C05452=1114.565,178.971,-64.399,-179.216,9.112,149.562
C05453=1114.569,178.722,-64.376,-179.219,9.109,149.562
C05454=1114.574,178.473,-64.352,-179.221,9.106,149.562
C05455=1114.579,178.224,-64.328,-179.223,9.103,149.562
C05456=1114.583,177.976,-64.304,-179.225,9.100,149.562
C05457=1114.588,177.727,-64.281,-179.228,9.097,149.562
C05458=1114.592,177.478,-64.257,-179.229,9.095,149.562
C05459=1114.597,177.229,-64.234,-179.232,9.091,149.562
C05460=1114.601,176.980,-64.210,-179.234,9.088,149.562
C05461=1114.606,176.732,-64.186,-179.236,9.086,149.561
C05462=1114.611,176.483,-64.163,-179.238,9.083,149.561
C05463=1114.615,176.233,-64.139,-179.241,9.079,149.561
C05464=1114.619,175.985,-64.115,-179.242,9.077,149.561
C05465=1114.624,175.736,-64.092,-179.245,9.074,149.561
C05466=1114.628,175.487,-64.068,-179.247,9.071,149.561
C05467=1114.633,175.238,-64.044,-179.249,9.068,149.561
C05468=1114.638,174.989,-64.021,-179.251,9.065,149.561
C05469=1114.642,174.740,-63.997,-179.253,9.062,149.561
C05470=1114.647,174.492,-63.973,-179.255,9.059,149.560
C05471=1114.651,174.243,-63.950,-179.258,9.056,149.560
C05472=1114.656,173.994,-63.927,-179.260,9.053,149.560
C05473=1114.661,173.745,-63.903,-179.262,9.050,149.560
C05474=1114.665,173.496,-63.879,-179.264,9.047,149.560
C05475=1114.670,173.247,-63.856,-179.267,9.044,149.560
C05476=1114.675,172.998,-63.833,-179.269,9.041,149.560
C05477=1114.678,172.749,-63.810,-179.271,9.038,149.560
C05478=1114.683,172.500,-63.786,-179.273,9.035,149.560
C05479=1114.687,172.287,-63.765,-179.275,9.032,149.560
C05480=1114.691,172.073,-63.745,-179.277,9.030,149.560
C05481=1114.695,171.860,-63.726,-179.278,9.027,149.559
C05482=1114.699,171.646,-63.706,-179.280,9.025,149.559
C05483=1114.703,171.432,-63.685,-179.282,9.023,149.559
C05484=1114.707,171.219,-63.666,-179.284,9.019,149.559
C05485=1114.711,171.005,-63.646,-179.286,9.017,149.559
C05486=1114.715,170.792,-63.626,-179.288,9.015,149.559
C05487=1114.719,170.543,-63.603,-179.290,9.011,149.559
C05488=1114.724,170.294,-63.579,-179.292,9.009,149.559
C05489=1114.728,170.045,-63.555,-179.295,9.006,149.559
C05490=1114.733,169.796,-63.532,-179.297,9.002,149.559
C05491=1114.737,169.548,-63.509,-179.299,8.999,149.559
C05492=1114.742,169.299,-63.486,-179.301,8.997,149.558
C05493=1114.747,169.050,-63.463,-179.303,8.993,149.558
C05494=1114.752,168.801,-63.439,-179.306,8.990,149.558
C05495=1114.756,168.552,-63.416,-179.308,8.987,149.558
C05496=1114.760,168.303,-63.393,-179.310,8.984,149.558
C05497=1114.765,168.054,-63.370,-179.312,8.981,149.558
C05498=1114.770,167.805,-63.347,-179.315,8.978,149.558
C05499=1114.774,167.557,-63.324,-179.317,8.975,149.558
C05500=1114.779,167.307,-63.301,-179.319,8.972,149.558
C05501=1114.784,167.059,-63.278,-179.321,8.969,149.558
C05502=1114.789,166.810,-63.255,-179.323,8.966,149.557
C05503=1114.793,166.561,-63.232,-179.326,8.963,149.557
C05504=1114.797,166.312,-63.209,-179.328,8.960,149.557
C05505=1114.802,166.063,-63.185,-179.330,8.957,149.557
C05506=1114.806,165.814,-63.163,-179.332,8.954,149.557
C05507=1114.811,165.566,-63.140,-179.335,8.951,149.557
C05508=1114.816,165.317,-63.116,-179.337,8.947,149.557
C05509=1114.820,165.067,-63.094,-179.339,8.945,149.557
C05510=1114.825,164.818,-63.071,-179.341,8.941,149.556
C05511=1114.830,164.569,-63.047,-179.343,8.938,149.556
C05512=1114.834,164.321,-63.025,-179.346,8.935,149.556
C05513=1114.839,164.072,-63.002,-179.348,8.932,149.556
C05514=1114.843,163.823,-62.980,-179.350,8.929,149.556
C05515=1114.848,163.574,-62.956,-179.352,8.926,149.556
C05516=1114.852,163.325,-62.934,-179.355,8.923,149.556
C05517=1114.857,163.076,-62.910,-179.357,8.919,149.556
C05518=1114.862,162.827,-62.888,-179.359,8.916,149.556
C05519=1114.866,162.579,-62.865,-179.362,8.913,149.555
C05520=1114.871,162.329,-62.842,-179.363,8.910,149.555
C05521=1114.875,162.080,-62.820,-179.366,8.907,149.555
C05522=1114.880,161.832,-62.797,-179.368,8.904,149.555
C05523=1114.884,161.583,-62.774,-179.370,8.901,149.555
C05524=1114.889,161.333,-62.751,-179.372,8.897,149.555
C05525=1114.893,161.085,-62.729,-179.375,8.894,149.555
C05526=1114.899,160.836,-62.706,-179.377,8.890,149.554
C05527=1114.903,160.587,-62.684,-179.379,8.888,149.554
C05528=1114.908,160.338,-62.660,-179.381,8.885,149.554
C05529=1114.912,160.089,-62.637,-179.383,8.882,149.554
C05530=1114.917,159.840,-62.615,-179.386,8.878,149.554
C05531=1114.921,159.592,-62.592,-179.388,8.875,149.554
C05532=1114.926,159.342,-62.570,-179.390,8.871,149.554
C05533=1114.930,159.093,-62.547,-179.393,8.868,149.554
C05534=1114.935,158.845,-62.525,-179.395,8.865,149.553
C05535=1114.939,158.631,-62.505,-179.397,8.862,149.553
C05536=1114.943,158.417,-62.486,-179.398,8.860,149.553
C05537=1114.947,158.203,-62.467,-179.401,8.857,149.553
C05538=1114.951,157.989,-62.448,-179.402,8.854,149.553
C05539=1114.955,157.776,-62.428,-179.405,8.851,149.553
C05540=1114.959,157.562,-62.409,-179.406,8.848,149.553
C05541=1114.963,157.349,-62.389,-179.408,8.846,149.553
C05542=1114.967,157.134,-62.370,-179.410,8.842,149.552
C05543=1114.972,156.886,-62.348,-179.413,8.839,149.552
C05544=1114.976,156.637,-62.326,-179.415,8.836,149.552
C05545=1114.981,156.388,-62.302,-179.417,8.833,149.552
C05546=1114.985,156.139,-62.281,-179.419,8.829,149.552
C05547=1114.990,155.890,-62.259,-179.421,8.826,149.552
C05548=1114.994,155.641,-62.235,-179.424,8.823,149.551
C05549=1114.999,155.392,-62.214,-179.425,8.820,149.551
C05550=1115.004,155.143,-62.191,-179.427,8.816,149.551
C05551=1115.008,154.894,-62.168,-179.430,8.813,149.551
C05552=1115.013,154.645,-62.146,-179.432,8.810,149.551
C05553=1115.017,154.396,-62.124,-179.435,8.805,149.551
C05554=1115.023,154.148,-62.101,-179.437,8.802,149.550
C05555=1115.027,153.898,-62.079,-179.439,8.799,149.550
C05556=1115.032,153.650,-62.058,-179.441,8.795,149.550
C05557=1115.036,153.400,-62.036,-179.443,8.792,149.550
C05558=1115.041,153.151,-62.012,-179.446,8.789,149.550
C05559=1115.046,152.903,-61.991,-179.448,8.785,149.550
C05560=1115.050,152.653,-61.969,-179.450,8.782,149.549
C05561=1115.055,152.405,-61.947,-179.452,8.778,149.549
C05562=1115.060,152.156,-61.923,-179.455,8.775,149.549
C05563=1115.064,151.907,-61.902,-179.457,8.772,149.549
C05564=1115.069,151.658,-61.880,-179.459,8.768,149.549
C05565=1115.074,151.409,-61.858,-179.461,8.765,149.548
C05566=1115.078,151.160,-61.836,-179.463,8.761,149.548
C05567=1115.083,150.910,-61.813,-179.466,8.758,149.548
C05568=1115.088,150.661,-61.792,-179.468,8.755,149.548
C05569=1115.092,150.412,-61.770,-179.470,8.750,149.548
C05570=1115.097,150.164,-61.747,-179.472,8.747,149.547
C05571=1115.101,149.915,-61.725,-179.475,8.743,149.547
C05572=1115.106,149.666,-61.704,-179.477,8.740,149.547
C05573=1115.111,149.417,-61.682,-179.479,8.736,149.547
C05574=1115.116,149.168,-61.659,-179.481,8.733,149.546
C05575=1115.120,148.919,-61.638,-179.483,8.729,149.546
C05576=1115.125,148.670,-61.615,-179.485,8.726,149.546
C05577=1115.130,148.421,-61.594,-179.488,8.722,149.546
C05578=1115.134,148.172,-61.572,-179.490,8.718,149.545
C05579=1115.139,147.923,-61.550,-179.492,8.715,149.545
C05580=1115.143,147.674,-61.528,-179.494,8.711,149.545
C05581=1115.148,147.425,-61.506,-179.496,8.708,149.545
C05582=1115.152,147.176,-61.484,-179.499,8.704,149.544
C05583=1115.157,146.927,-61.463,-179.501,8.700,149.544
C05584=1115.162,146.677,-61.441,-179.503,8.697,149.544
C05585=1115.166,146.429,-61.420,-179.505,8.693,149.544
C05586=1115.171,146.180,-61.398,-179.507,8.690,149.544
C05587=1115.176,145.931,-61.376,-179.510,8.685,149.543
C05588=1115.180,145.682,-61.354,-179.512,8.682,149.543
C05589=1115.185,145.433,-61.332,-179.514,8.678,149.543
C05590=1115.190,145.184,-61.310,-179.516,8.675,149.543
C05591=1115.194,144.970,-61.291,-179.518,8.671,149.542
C05592=1115.198,144.756,-61.274,-179.519,8.668,149.542
C05593=1115.202,144.542,-61.255,-179.520,8.666,149.542
C05594=1115.206,144.329,-61.237,-179.521,8.662,149.541
C05595=1115.210,144.114,-61.218,-179.523,8.660,149.541
C05596=1115.213,143.901,-61.199,-179.524,8.657,149.541
C05597=1115.218,143.687,-61.180,-179.525,8.654,149.540
C05598=1115.221,143.473,-61.162,-179.527,8.651,149.540
C05599=1115.226,143.225,-61.140,-179.529,8.648,149.540
C05600=1115.231,142.975,-61.119,-179.531,8.644,149.539
C05601=1115.236,142.726,-61.097,-179.532,8.641,149.539
C05602=1115.241,142.477,-61.076,-179.534,8.637,149.539
C05603=1115.245,142.227,-61.054,-179.536,8.634,149.539
C05604=1115.250,141.979,-61.033,-179.537,8.631,149.538
C05605=1115.255,141.730,-61.011,-179.539,8.627,149.538
C05606=1115.259,141.480,-60.990,-179.540,8.623,149.537
C05607=1115.264,141.232,-60.968,-179.542,8.621,149.537
C05608=1115.268,140.983,-60.947,-179.544,8.617,149.537
C05609=1115.273,140.733,-60.925,-179.545,8.614,149.537
C05610=1115.278,140.485,-60.904,-179.547,8.610,149.536
C05611=1115.283,140.236,-60.882,-179.549,8.607,149.536
C05612=1115.287,139.986,-60.861,-179.550,8.604,149.536
C05613=1115.291,139.738,-60.840,-179.552,8.600,149.535
C05614=1115.297,139.488,-60.819,-179.554,8.597,149.535
C05615=1115.301,139.240,-60.797,-179.555,8.594,149.535
C05616=1115.306,138.990,-60.775,-179.557,8.590,149.534
C05617=1115.310,138.741,-60.755,-179.559,8.587,149.534
C05618=1115.315,138.493,-60.733,-179.560,8.583,149.534
C05619=1115.320,138.243,-60.712,-179.562,8.580,149.533
C05620=1115.324,137.994,-60.690,-179.563,8.577,149.533
C05621=1115.329,137.745,-60.669,-179.565,8.573,149.533
C05622=1115.334,137.497,-60.648,-179.567,8.570,149.533
C05623=1115.338,137.247,-60.626,-179.568,8.567,149.532
C05624=1115.343,136.998,-60.605,-179.570,8.563,149.532
C05625=1115.348,136.749,-60.584,-179.572,8.560,149.532
C05626=1115.353,136.500,-60.563,-179.573,8.557,149.531
C05627=1115.357,136.250,-60.541,-179.575,8.553,149.531
C05628=1115.361,136.002,-60.520,-179.578,8.550,149.531
C05629=1115.366,135.753,-60.499,-179.579,8.547,149.530
C05630=1115.372,135.504,-60.478,-179.581,8.543,149.530
C05631=1115.376,135.255,-60.457,-179.583,8.540,149.530
C05632=1115.380,135.005,-60.436,-179.584,8.537,149.529
C05633=1115.385,134.757,-60.414,-179.586,8.533,149.529
C05634=1115.390,134.507,-60.393,-179.587,8.530,149.529
C05635=1115.395,134.258,-60.373,-179.589,8.527,149.529
C05636=1115.400,134.010,-60.351,-179.591,8.523,149.528
C05637=1115.404,133.760,-60.330,-179.592,8.520,149.528
C05638=1115.409,133.511,-60.310,-179.594,8.516,149.528
C05639=1115.414,133.262,-60.288,-179.596,8.513,149.527
C05640=1115.418,133.013,-60.267,-179.598,8.510,149.527
C05641=1115.423,132.764,-60.247,-179.599,8.506,149.527
C05642=1115.428,132.515,-60.225,-179.601,8.503,149.526
C05643=1115.432,132.266,-60.204,-179.603,8.500,149.526
C05644=1115.437,132.017,-60.183,-179.605,8.497,149.526
C05645=1115.441,131.768,-60.163,-179.606,8.493,149.526
C05646=1115.446,131.519,-60.141,-179.608,8.490,149.525
C05647=1115.451,131.305,-60.124,-179.609,8.487,149.525
C05648=1115.454,131.091,-60.106,-179.611,8.484,149.525
C05649=1115.459,130.877,-60.087,-179.613,8.481,149.525
C05650=1115.463,130.663,-60.069,-179.614,8.478,149.524
C05651=1115.467,130.449,-60.052,-179.616,8.476,149.524
C05652=1115.470,130.235,-60.034,-179.617,8.473,149.524
C05653=1115.474,130.021,-60.016,-179.618,8.470,149.524
C05654=1115.479,129.807,-59.998,-179.620,8.467,149.523
C05655=1115.484,129.558,-59.978,-179.622,8.464,149.523
C05656=1115.488,129.309,-59.956,-179.624,8.460,149.523
C05657=1115.493,129.060,-59.935,-179.625,8.457,149.522
C05658=1115.498,128.811,-59.914,-179.627,8.454,149.522
C05659=1115.502,128.562,-59.894,-179.629,8.450,149.522
C05660=1115.507,128.312,-59.873,-179.630,8.447,149.522
C05661=1115.512,128.063,-59.853,-179.632,8.444,149.521
C05662=1115.517,127.814,-59.832,-179.634,8.440,149.521
C05663=1115.521,127.565,-59.811,-179.635,8.437,149.521
C05664=1115.527,127.316,-59.790,-179.637,8.434,149.521
C05665=1115.531,127.067,-59.770,-179.639,8.430,149.520
C05666=1115.535,126.818,-59.750,-179.641,8.427,149.520
C05667=1115.541,126.569,-59.729,-179.643,8.424,149.520
C05668=1115.545,126.320,-59.708,-179.645,8.420,149.520
C05669=1115.550,126.071,-59.687,-179.646,8.418,149.519
C05670=1115.555,125.822,-59.667,-179.648,8.414,149.519
C05671=1115.559,125.573,-59.647,-179.650,8.410,149.519
C05672=1115.564,125.323,-59.626,-179.652,8.407,149.518
C05673=1115.569,125.075,-59.605,-179.653,8.404,149.518
C05674=1115.573,124.825,-59.584,-179.655,8.400,149.518
C05675=1115.578,124.576,-59.563,-179.657,8.397,149.518
C05676=1115.582,124.327,-59.543,-179.658,8.394,149.517
C05677=1115.587,124.077,-59.522,-179.660,8.390,149.517
C05678=1115.592,123.828,-59.502,-179.662,8.386,149.517
C05679=1115.596,123.580,-59.481,-179.664,8.384,149.516
C05680=1115.601,123.330,-59.460,-179.666,8.380,149.516
C05681=1115.606,123.081,-59.440,-179.668,8.377,149.516
C05682=1115.611,122.833,-59.420,-179.669,8.373,149.516
C05683=1115.616,122.583,-59.400,-179.671,8.370,149.515
C05684=1115.621,122.334,-59.379,-179.673,8.367,149.515
C05685=1115.625,122.085,-59.359,-179.675,8.363,149.515
C05686=1115.630,121.836,-59.339,-179.676,8.360,149.515
C05687=1115.635,121.587,-59.318,-179.678,8.357,149.514
C05688=1115.640,121.338,-59.298,-179.680,8.353,149.514
C05689=1115.644,121.089,-59.278,-179.682,8.350,149.514
C05690=1115.648,120.840,-59.257,-179.684,8.347,149.514
C05691=1115.654,120.590,-59.236,-179.685,8.343,149.513
C05692=1115.658,120.341,-59.216,-179.687,8.339,149.513
C05693=1115.663,120.092,-59.196,-179.689,8.337,149.513
C05694=1115.667,119.843,-59.176,-179.691,8.333,149.512
C05695=1115.672,119.594,-59.155,-179.692,8.329,149.512
C05696=1115.677,119.344,-59.135,-179.694,8.326,149.512
C05697=1115.682,119.095,-59.115,-179.696,8.323,149.512
C05698=1115.687,118.847,-59.095,-179.698,8.320,149.511
C05699=1115.691,118.597,-59.075,-179.700,8.316,149.511
C05700=1115.696,118.348,-59.055,-179.702,8.312,149.511
C05701=1115.701,118.099,-59.034,-179.703,8.310,149.510
C05702=1115.706,117.850,-59.014,-179.705,8.306,149.510
C05703=1115.710,117.636,-58.997,-179.707,8.303,149.510
C05704=1115.714,117.422,-58.979,-179.709,8.300,149.510
C05705=1115.717,117.208,-58.962,-179.710,8.297,149.509
C05706=1115.721,116.994,-58.945,-179.711,8.294,149.509
C05707=1115.726,116.780,-58.928,-179.712,8.291,149.509
C05708=1115.730,116.566,-58.911,-179.714,8.289,149.509
C05709=1115.734,116.351,-58.893,-179.716,8.285,149.508
C05710=1115.738,116.137,-58.876,-179.717,8.282,149.508
C05711=1115.743,115.888,-58.856,-179.719,8.279,149.508
C05712=1115.748,115.640,-58.836,-179.720,8.276,149.508
C05713=1115.753,115.390,-58.816,-179.722,8.272,149.507
C05714=1115.757,115.141,-58.796,-179.725,8.269,149.507
C05715=1115.762,114.892,-58.776,-179.727,8.265,149.507
C05716=1115.766,114.643,-58.756,-179.728,8.261,149.506
C05717=1115.771,114.393,-58.736,-179.730,8.259,149.506
C05718=1115.776,114.145,-58.716,-179.732,8.255,149.506
C05719=1115.781,113.895,-58.697,-179.734,8.252,149.506
C05720=1115.786,113.646,-58.676,-179.735,8.248,149.505
C05721=1115.791,113.396,-58.656,-179.737,8.244,149.505
C05722=1115.795,113.147,-58.636,-179.739,8.242,149.505
C05723=1115.800,112.899,-58.616,-179.740,8.238,149.504
C05724=1115.805,112.649,-58.597,-179.743,8.234,149.504
C05725=1115.810,112.400,-58.576,-179.745,8.231,149.504
C05726=1115.814,112.151,-58.557,-179.746,8.227,149.504
C05727=1115.820,111.902,-58.537,-179.748,8.224,149.503
C05728=1115.824,111.653,-58.517,-179.750,8.221,149.503
C05729=1115.829,111.403,-58.497,-179.751,8.217,149.503
C05730=1115.833,111.154,-58.477,-179.753,8.213,149.502
C05731=1115.839,110.905,-58.458,-179.755,8.210,149.502
C05732=1115.843,110.656,-58.439,-179.758,8.206,149.502
C05733=1115.847,110.406,-58.419,-179.760,8.203,149.502
C05734=1115.852,110.158,-58.399,-179.762,8.198,149.502
C05735=1115.857,109.909,-58.379,-179.764,8.195,149.501
C05736=1115.862,109.659,-58.360,-179.766,8.191,149.501
C05737=1115.867,109.410,-58.340,-179.768,8.188,149.501
C05738=1115.872,109.161,-58.320,-179.770,8.184,149.500
C05739=1115.876,108.912,-58.300,-179.773,8.180,149.500
C05740=1115.881,108.662,-58.281,-179.775,8.176,149.500
C05741=1115.887,108.413,-58.261,-179.776,8.172,149.500
C05742=1115.890,108.165,-58.242,-179.778,8.169,149.499
C05743=1115.895,107.915,-58.222,-179.781,8.165,149.499
C05744=1115.900,107.666,-58.203,-179.783,8.161,149.499
C05745=1115.905,107.417,-58.183,-179.785,8.157,149.498
C05746=1115.910,107.167,-58.163,-179.787,8.154,149.498
C05747=1115.915,106.918,-58.144,-179.788,8.150,149.498
C05748=1115.919,106.669,-58.125,-179.791,8.146,149.498
C05749=1115.924,106.419,-58.105,-179.793,8.142,149.497
C05750=1115.929,106.171,-58.085,-179.795,8.138,149.497
C05751=1115.934,105.922,-58.066,-179.797,8.135,149.497
C05752=1115.938,105.672,-58.047,-179.799,8.131,149.496
C05753=1115.943,105.423,-58.027,-179.801,8.127,149.496
C05754=1115.948,105.174,-58.008,-179.803,8.124,149.496
C05755=1115.953,104.925,-57.988,-179.804,8.120,149.495
C05756=1115.957,104.676,-57.969,-179.807,8.116,149.495
C05757=1115.962,104.426,-57.950,-179.808,8.112,149.495
C05758=1115.967,104.177,-57.930,-179.811,8.108,149.494
C05759=1115.971,103.963,-57.914,-179.812,8.105,149.494
C05760=1115.976,103.749,-57.897,-179.814,8.102,149.494
C05761=1115.980,103.534,-57.881,-179.815,8.099,149.494
C05762=1115.984,103.321,-57.864,-179.817,8.095,149.493
C05763=1115.988,103.107,-57.847,-179.818,8.092,149.493
C05764=1115.992,102.892,-57.831,-179.820,8.089,149.493
C05765=1115.996,102.678,-57.815,-179.822,8.085,149.492
C05766=1116.000,102.464,-57.798,-179.823,8.082,149.492
C05767=1116.005,102.214,-57.779,-179.825,8.078,149.492
C05768=1116.010,101.966,-57.760,-179.827,8.075,149.491
C05769=1116.015,101.716,-57.740,-179.828,8.071,149.491
C05770=1116.020,101.467,-57.721,-179.830,8.067,149.491
C05771=1116.024,101.218,-57.702,-179.832,8.064,149.490
C05772=1116.029,100.969,-57.683,-179.834,8.059,149.490
C05773=1116.034,100.719,-57.664,-179.836,8.055,149.489
C05774=1116.039,100.470,-57.645,-179.837,8.051,149.489
C05775=1116.044,100.221,-57.625,-179.840,8.048,149.489
C05776=1116.048,99.972,-57.607,-179.841,8.044,149.488
C05777=1116.053,99.723,-57.587,-179.843,8.040,149.488
C05778=1116.058,99.474,-57.569,-179.844,8.036,149.488
C05779=1116.063,99.224,-57.549,-179.846,8.032,149.487
C05780=1116.067,98.975,-57.531,-179.848,8.029,149.487
C05781=1116.072,98.725,-57.512,-179.850,8.025,149.486
C05782=1116.078,98.476,-57.493,-179.851,8.021,149.486
C05783=1116.082,98.227,-57.473,-179.853,8.017,149.486
C05784=1116.087,97.978,-57.454,-179.854,8.013,149.485
C05785=1116.091,97.728,-57.436,-179.856,8.009,149.485
C05786=1116.097,97.480,-57.417,-179.858,8.006,149.484
C05787=1116.101,97.230,-57.397,-179.860,8.002,149.484
C05788=1116.106,96.981,-57.379,-179.861,7.998,149.484
C05789=1116.110,96.732,-57.360,-179.863,7.994,149.483
C05790=1116.116,96.482,-57.341,-179.864,7.990,149.483
C05791=1116.121,96.234,-57.323,-179.866,7.986,149.482
C05792=1116.125,95.984,-57.304,-179.868,7.982,149.482
C05793=1116.130,95.735,-57.285,-179.869,7.978,149.481
C05794=1116.134,95.486,-57.266,-179.871,7.974,149.481
C05795=1116.140,95.236,-57.247,-179.872,7.971,149.481
C05796=1116.144,94.987,-57.229,-179.874,7.967,149.480
C05797=1116.150,94.737,-57.210,-179.875,7.964,149.480
C05798=1116.154,94.489,-57.191,-179.877,7.960,149.479
C05799=1116.159,94.239,-57.171,-179.878,7.956,149.479
C05800=1116.164,93.990,-57.153,-179.880,7.952,149.478
C05801=1116.168,93.741,-57.135,-179.881,7.948,149.478
C05802=1116.173,93.491,-57.116,-179.883,7.944,149.478
C05803=1116.178,93.242,-57.098,-179.885,7.940,149.477
C05804=1116.183,92.994,-57.079,-179.886,7.936,149.476
C05805=1116.188,92.743,-57.060,-179.887,7.932,149.476
C05806=1116.193,92.495,-57.041,-179.889,7.928,149.476
C05807=1116.198,92.245,-57.023,-179.890,7.925,149.475
C05808=1116.202,91.996,-57.004,-179.892,7.921,149.475
C05809=1116.207,91.747,-56.986,-179.893,7.917,149.474
C05810=1116.213,91.497,-56.967,-179.895,7.913,149.474
C05811=1116.217,91.248,-56.948,-179.896,7.909,149.473
C05812=1116.222,90.999,-56.930,-179.897,7.905,149.473
C05813=1116.226,90.750,-56.911,-179.899,7.901,149.472
C05814=1116.231,90.500,-56.893,-179.900,7.898,149.472
C05815=1116.235,90.286,-56.876,-179.902,7.894,149.472
C05816=1116.240,90.072,-56.861,-179.903,7.891,149.471
C05817=1116.244,89.858,-56.845,-179.904,7.888,149.471
C05818=1116.248,89.644,-56.829,-179.905,7.885,149.470
C05819=1116.252,89.429,-56.813,-179.906,7.881,149.470
C05820=1116.256,89.215,-56.797,-179.907,7.878,149.469
C05821=1116.261,89.001,-56.781,-179.908,7.875,149.469
C05822=1116.265,88.787,-56.766,-179.910,7.871,149.468
C05823=1116.270,88.537,-56.748,-179.911,7.868,149.468
C05824=1116.274,88.288,-56.729,-179.912,7.864,149.468
C05825=1116.279,88.039,-56.710,-179.914,7.860,149.467
C05826=1116.284,87.790,-56.692,-179.915,7.856,149.467
C05827=1116.289,87.540,-56.674,-179.916,7.853,149.466
C05828=1116.293,87.291,-56.655,-179.918,7.849,149.466
C05829=1116.298,87.042,-56.637,-179.919,7.845,149.465
C05830=1116.304,86.792,-56.619,-179.920,7.841,149.465
C05831=1116.309,86.543,-56.601,-179.921,7.838,149.464
C05832=1116.313,86.293,-56.582,-179.922,7.833,149.464
C05833=1116.318,86.045,-56.564,-179.924,7.829,149.463
C05834=1116.323,85.796,-56.546,-179.925,7.826,149.463
C05835=1116.328,85.546,-56.527,-179.926,7.822,149.462
C05836=1116.332,85.296,-56.509,-179.928,7.818,149.462
C05837=1116.337,85.047,-56.491,-179.928,7.815,149.461
C05838=1116.342,84.798,-56.473,-179.930,7.811,149.461
C05839=1116.347,84.549,-56.455,-179.931,7.807,149.460
C05840=1116.352,84.300,-56.437,-179.932,7.803,149.459
C05841=1116.356,84.050,-56.418,-179.933,7.799,149.459
C05842=1116.361,83.801,-56.400,-179.935,7.795,149.458
C05843=1116.366,83.552,-56.382,-179.936,7.792,149.458
C05844=1116.372,83.302,-56.363,-179.937,7.788,149.457
C05845=1116.377,83.053,-56.345,-179.938,7.784,149.457
C05846=1116.381,82.803,-56.327,-179.939,7.781,149.456
C05847=1116.386,82.554,-56.309,-179.940,7.776,149.456
C05848=1116.391,82.305,-56.291,-179.941,7.773,149.455
C05849=1116.396,82.056,-56.273,-179.942,7.769,149.455
C05850=1116.400,81.807,-56.255,-179.944,7.765,149.454
C05851=1116.405,81.558,-56.237,-179.945,7.762,149.454
C05852=1116.410,81.308,-56.219,-179.946,7.758,149.453
C05853=1116.415,81.058,-56.201,-179.947,7.754,149.453
C05854=1116.420,80.809,-56.183,-179.948,7.750,149.452
C05855=1116.424,80.560,-56.165,-179.949,7.747,149.451
C05856=1116.429,80.311,-56.147,-179.950,7.743,149.451
C05857=1116.434,80.062,-56.129,-179.951,7.739,149.450
C05858=1116.439,79.813,-56.111,-179.952,7.736,149.450
C05859=1116.444,79.563,-56.094,-179.954,7.731,149.449
C05860=1116.449,79.314,-56.076,-179.954,7.728,149.449
C05861=1116.454,79.064,-56.057,-179.956,7.724,149.448
C05862=1116.459,78.815,-56.039,-179.956,7.720,149.448
C05863=1116.463,78.565,-56.021,-179.958,7.716,149.447
C05864=1116.468,78.316,-56.003,-179.958,7.713,149.447
C05865=1116.473,78.067,-55.985,-179.959,7.710,149.446
C05866=1116.478,77.818,-55.967,-179.960,7.706,149.445
C05867=1116.483,77.568,-55.950,-179.961,7.702,149.445
C05868=1116.488,77.319,-55.932,-179.962,7.698,149.444
C05869=1116.493,77.070,-55.914,-179.963,7.695,149.444
C05870=1116.498,76.821,-55.896,-179.964,7.691,149.443
C05871=1116.504,76.515,-55.874,-179.966,7.686,149.443
C05872=1116.510,76.208,-55.853,-179.967,7.681,149.442
C05873=1116.516,75.902,-55.831,-179.969,7.676,149.441
C05874=1116.522,75.596,-55.809,-179.971,7.672,149.441
C05875=1116.527,75.347,-55.791,-179.972,7.667,149.440
C05876=1116.532,75.097,-55.774,-179.974,7.664,149.440
C05877=1116.536,74.849,-55.756,-179.976,7.660,149.439
C05878=1116.541,74.599,-55.738,-179.977,7.656,149.439
C05879=1116.546,74.350,-55.720,-179.978,7.651,149.438
C05880=1116.551,74.100,-55.703,-179.980,7.648,149.438
C05881=1116.556,73.851,-55.685,-179.981,7.644,149.437
C05882=1116.561,73.602,-55.667,-179.983,7.640,149.437
C05883=1116.566,73.353,-55.651,-179.984,7.635,149.436
C05884=1116.570,73.103,-55.633,-179.985,7.632,149.436
C05885=1116.575,72.854,-55.615,-179.987,7.628,149.436
C05886=1116.581,72.604,-55.597,-179.988,7.624,149.435
C05887=1116.586,72.355,-55.579,-179.989,7.620,149.434
C05888=1116.590,72.106,-55.563,-179.991,7.616,149.434
C05889=1116.595,71.857,-55.545,-179.992,7.612,149.434
C05890=1116.600,71.607,-55.527,-179.994,7.608,149.433
C05891=1116.605,71.358,-55.509,-179.995,7.604,149.432
C05892=1116.609,71.109,-55.492,-179.997,7.600,149.432
C05893=1116.614,70.859,-55.475,-179.998,7.596,149.431
C05894=1116.619,70.610,-55.457,-179.999,7.592,149.431
C05895=1116.625,70.360,-55.440,179.999,7.588,149.431
C05896=1116.629,70.111,-55.422,179.997,7.584,149.430
C05897=1116.634,69.861,-55.405,179.997,7.581,149.429
C05898=1116.639,69.612,-55.387,179.995,7.577,149.429
C05899=1116.644,69.362,-55.370,179.994,7.573,149.429
C05900=1116.648,69.114,-55.352,179.993,7.569,149.428
C05901=1116.654,68.864,-55.335,179.991,7.565,149.428
C05902=1116.659,68.615,-55.317,179.990,7.561,149.427
C05903=1116.663,68.366,-55.301,179.988,7.557,149.426
C05904=1116.668,68.117,-55.283,179.987,7.553,149.426
C05905=1116.674,67.867,-55.265,179.985,7.549,149.426
C05906=1116.678,67.617,-55.249,179.984,7.545,149.425
C05907=1116.683,67.368,-55.231,179.983,7.541,149.425
C05908=1116.687,67.119,-55.214,179.982,7.538,149.424
C05909=1116.692,66.870,-55.196,179.981,7.533,149.423
C05910=1116.698,66.620,-55.179,179.979,7.529,149.423
C05911=1116.705,66.249,-55.153,179.977,7.523,149.422
C05912=1116.713,65.876,-55.128,179.975,7.517,149.421
C05913=1116.720,65.504,-55.102,179.973,7.511,149.421
C05914=1116.727,65.132,-55.076,179.971,7.505,149.420
C05915=1116.732,64.882,-55.059,179.970,7.502,149.420
C05916=1116.737,64.634,-55.043,179.968,7.498,149.419
C05917=1116.742,64.384,-55.025,179.967,7.494,149.418
C05918=1116.746,64.135,-55.008,179.966,7.490,149.418
C05919=1116.751,63.885,-54.991,179.964,7.486,149.417
C05920=1116.756,63.636,-54.974,179.963,7.482,149.417
C05921=1116.761,63.387,-54.957,179.962,7.477,149.416
C05922=1116.766,63.138,-54.940,179.960,7.474,149.416
C05923=1116.770,62.922,-54.925,179.959,7.470,149.415
C05924=1116.775,62.708,-54.910,179.958,7.467,149.415
C05925=1116.778,62.494,-54.896,179.957,7.463,149.415
C05926=1116.784,62.279,-54.881,179.956,7.460,149.414
C05927=1116.787,62.066,-54.867,179.955,7.457,149.414
C05928=1116.792,61.851,-54.851,179.954,7.453,149.413
C05929=1116.796,61.637,-54.838,179.953,7.450,149.413
C05930=1116.800,61.422,-54.822,179.952,7.447,149.412
C05931=1116.805,61.172,-54.806,179.950,7.443,149.412
C05932=1116.810,60.924,-54.789,179.949,7.438,149.411
C05933=1116.815,60.674,-54.772,179.947,7.434,149.411
C05934=1116.819,60.424,-54.755,179.946,7.431,149.410
C05935=1116.825,60.174,-54.738,179.945,7.426,149.410
C05936=1116.830,59.926,-54.722,179.943,7.422,149.409
C05937=1116.835,59.676,-54.705,179.942,7.418,149.409
C05938=1116.839,59.427,-54.687,179.941,7.414,149.408
C05939=1116.844,59.178,-54.671,179.940,7.411,149.407
C05940=1116.849,58.928,-54.654,179.938,7.407,149.407
C05941=1116.854,58.679,-54.637,179.937,7.403,149.407
C05942=1116.859,58.429,-54.620,179.936,7.399,149.406
C05943=1116.864,58.180,-54.603,179.934,7.395,149.406
C05944=1116.869,57.931,-54.587,179.933,7.390,149.405
C05945=1116.874,57.681,-54.569,179.932,7.386,149.404
C05946=1116.879,57.432,-54.553,179.931,7.382,149.404
C05947=1116.883,57.183,-54.536,179.929,7.378,149.403
C05948=1116.889,56.933,-54.519,179.928,7.375,149.403
C05949=1116.894,56.684,-54.504,179.927,7.371,149.402
C05950=1116.898,56.434,-54.487,179.926,7.367,149.402
C05951=1116.904,56.184,-54.470,179.924,7.363,149.401
C05952=1116.909,55.936,-54.453,179.923,7.358,149.401
C05953=1116.913,55.686,-54.437,179.922,7.354,149.400
C05954=1116.918,55.436,-54.419,179.921,7.350,149.399
C05955=1116.923,55.188,-54.403,179.919,7.346,149.399
C05956=1116.928,54.938,-54.386,179.918,7.343,149.398
C05957=1116.932,54.689,-54.370,179.917,7.339,149.398
C05958=1116.939,54.439,-54.354,179.916,7.334,149.397
C05959=1116.943,54.189,-54.337,179.914,7.331,149.397
C05960=1116.948,53.941,-54.321,179.913,7.326,149.396
C05961=1116.953,53.691,-54.304,179.912,7.322,149.396
C05962=1116.958,53.441,-54.287,179.911,7.318,149.395
C05963=1116.963,53.193,-54.270,179.909,7.314,149.395
C05964=1116.968,52.942,-54.254,179.909,7.311,149.394
C05965=1116.973,52.694,-54.238,179.907,7.306,149.393
C05966=1116.978,52.444,-54.221,179.906,7.302,149.393
C05967=1116.982,52.194,-54.204,179.905,7.298,149.392
C05968=1116.988,51.945,-54.189,179.903,7.294,149.392
C05969=1116.992,51.695,-54.172,179.902,7.290,149.391
C05970=1116.997,51.447,-54.156,179.901,7.286,149.391
C05971=1117.003,51.197,-54.138,179.900,7.282,149.390
C05972=1117.008,50.947,-54.123,179.899,7.278,149.390
C05973=1117.013,50.698,-54.106,179.897,7.274,149.389
C05974=1117.017,50.448,-54.089,179.896,7.270,149.388
C05975=1117.022,50.199,-54.074,179.895,7.266,149.388
C05976=1117.027,49.950,-54.057,179.894,7.262,149.387
C05977=1117.032,49.701,-54.041,179.893,7.257,149.387
C05978=1117.037,49.451,-54.025,179.891,7.254,149.386
C05979=1117.042,49.236,-54.011,179.890,7.250,149.386
C05980=1117.046,49.022,-53.997,179.890,7.247,149.385
C05981=1117.049,48.807,-53.982,179.888,7.243,149.385
C05982=1117.054,48.593,-53.968,179.887,7.240,149.384
C05983=1117.058,48.379,-53.955,179.887,7.236,149.384
C05984=1117.063,48.164,-53.940,179.885,7.232,149.383
C05985=1117.067,47.949,-53.926,179.884,7.229,149.383
C05986=1117.071,47.735,-53.913,179.883,7.226,149.382
C05987=1117.076,47.486,-53.896,179.882,7.222,149.382
C05988=1117.081,47.236,-53.880,179.881,7.218,149.381
C05989=1117.086,46.987,-53.864,179.880,7.214,149.381
C05990=1117.091,46.737,-53.848,179.879,7.209,149.380
C05991=1117.096,46.488,-53.832,179.877,7.205,149.379
C05992=1117.101,46.238,-53.816,179.876,7.201,149.379
C05993=1117.106,45.989,-53.800,179.875,7.198,149.378
C05994=1117.111,45.739,-53.784,179.874,7.193,149.378
C05995=1117.116,45.490,-53.767,179.873,7.189,149.377
C05996=1117.120,45.240,-53.751,179.872,7.185,149.377
C05997=1117.125,44.991,-53.735,179.871,7.181,149.376
C05998=1117.131,44.742,-53.719,179.870,7.176,149.375
C05999=1117.136,44.492,-53.704,179.868,7.173,149.375
C06000=1117.141,44.243,-53.687,179.867,7.168,149.374
C06001=1117.146,43.993,-53.671,179.867,7.165,149.374
C06002=1117.151,43.744,-53.655,179.865,7.161,149.373
C06003=1117.155,43.494,-53.639,179.864,7.157,149.372
C06004=1117.161,43.245,-53.623,179.863,7.152,149.372
C06005=1117.166,42.996,-53.607,179.862,7.148,149.371
C06006=1117.171,42.746,-53.591,179.860,7.144,149.371
C06007=1117.176,42.497,-53.575,179.859,7.140,149.370
C06008=1117.181,42.247,-53.559,179.858,7.135,149.369
C06009=1117.186,41.998,-53.543,179.858,7.132,149.369
C06010=1117.190,41.749,-53.528,179.857,7.128,149.368
C06011=1117.195,41.499,-53.512,179.855,7.124,149.368
C06012=1117.200,41.250,-53.496,179.854,7.119,149.367
C06013=1117.205,41.000,-53.480,179.853,7.115,149.366
C06014=1117.210,40.751,-53.464,179.852,7.111,149.366
C06015=1117.216,40.501,-53.448,179.851,7.106,149.365
C06016=1117.220,40.251,-53.432,179.849,7.103,149.365
C06017=1117.226,40.002,-53.416,179.849,7.099,149.364
C06018=1117.230,39.753,-53.401,179.848,7.095,149.363
C06019=1117.235,39.503,-53.385,179.847,7.090,149.363
C06020=1117.240,39.254,-53.369,179.845,7.086,149.362
C06021=1117.246,39.004,-53.354,179.844,7.082,149.361
C06022=1117.250,38.755,-53.337,179.843,7.078,149.361
C06023=1117.255,38.506,-53.322,179.842,7.074,149.360
C06024=1117.260,38.256,-53.307,179.841,7.069,149.360
C06025=1117.265,38.006,-53.291,179.840,7.065,149.359
C06026=1117.270,37.757,-53.275,179.839,7.061,149.358
C06027=1117.276,37.508,-53.259,179.838,7.057,149.358
C06028=1117.280,37.258,-53.243,179.837,7.053,149.357
C06029=1117.285,37.009,-53.228,179.836,7.048,149.356
C06030=1117.290,36.760,-53.212,179.834,7.045,149.356
C06031=1117.296,36.510,-53.197,179.833,7.040,149.355
C06032=1117.300,36.260,-53.181,179.832,7.036,149.355
C06033=1117.305,36.011,-53.166,179.831,7.032,149.354
C06034=1117.311,35.762,-53.150,179.831,7.028,149.353
C06035=1117.315,35.547,-53.136,179.830,7.024,149.353
C06036=1117.319,35.332,-53.123,179.829,7.021,149.352
C06037=1117.324,35.118,-53.110,179.828,7.017,149.352
C06038=1117.327,34.903,-53.096,179.827,7.013,149.351
C06039=1117.331,34.688,-53.083,179.826,7.010,149.351
C06040=1117.336,34.474,-53.070,179.825,7.006,149.350
C06041=1117.340,34.259,-53.057,179.824,7.002,149.349
C06042=1117.344,34.045,-53.043,179.824,6.999,149.349
C06043=1117.350,33.795,-53.027,179.822,6.995,149.348
C06044=1117.355,33.546,-53.012,179.821,6.991,149.348
C06045=1117.360,33.297,-52.997,179.820,6.986,149.347
C06046=1117.365,33.047,-52.981,179.819,6.982,149.346
C06047=1117.369,32.798,-52.966,179.818,6.978,149.346
C06048=1117.375,32.548,-52.950,179.817,6.973,149.345
C06049=1117.380,32.299,-52.935,179.817,6.970,149.344
C06050=1117.384,32.048,-52.920,179.816,6.965,149.344
C06051=1117.390,31.799,-52.904,179.815,6.961,149.343
C06052=1117.394,31.550,-52.889,179.814,6.956,149.342
C06053=1117.400,31.301,-52.874,179.813,6.952,149.342
C06054=1117.405,31.051,-52.858,179.812,6.948,149.341
C06055=1117.410,30.802,-52.843,179.811,6.944,149.340
C06056=1117.415,30.552,-52.827,179.810,6.939,149.340
C06057=1117.419,30.303,-52.812,179.809,6.935,149.339
C06058=1117.425,30.053,-52.797,179.808,6.931,149.338
C06059=1117.430,29.804,-52.782,179.807,6.927,149.338
C06060=1117.435,29.554,-52.767,179.806,6.923,149.337
C06061=1117.440,29.305,-52.751,179.805,6.918,149.336
C06062=1117.445,29.055,-52.736,179.804,6.914,149.336
C06063=1117.450,28.806,-52.720,179.803,6.910,149.335
C06064=1117.455,28.556,-52.706,179.802,6.905,149.334
C06065=1117.460,28.307,-52.690,179.801,6.901,149.334
C06066=1117.465,28.058,-52.675,179.800,6.896,149.333
C06067=1117.470,27.808,-52.660,179.799,6.892,149.332
C06068=1117.475,27.558,-52.645,179.798,6.888,149.332
C06069=1117.480,27.308,-52.630,179.798,6.884,149.331
C06070=1117.485,27.059,-52.615,179.797,6.880,149.330
C06071=1117.490,26.810,-52.599,179.796,6.875,149.329
C06072=1117.495,26.560,-52.585,179.795,6.871,149.329
C06073=1117.500,26.311,-52.569,179.794,6.867,149.328
C06074=1117.505,26.062,-52.554,179.793,6.862,149.327
C06075=1117.511,25.812,-52.539,179.792,6.858,149.327
C06076=1117.515,25.562,-52.524,179.791,6.853,149.326
C06077=1117.520,25.313,-52.509,179.790,6.849,149.325
C06078=1117.526,25.063,-52.494,179.789,6.845,149.325
C06079=1117.530,24.814,-52.479,179.788,6.840,149.324
C06080=1117.535,24.564,-52.463,179.788,6.836,149.323
C06081=1117.540,24.314,-52.449,179.787,6.832,149.322
C06082=1117.545,24.065,-52.434,179.786,6.828,149.322
C06083=1117.550,23.815,-52.419,179.785,6.824,149.321
C06084=1117.555,23.566,-52.404,179.784,6.819,149.320
C06085=1117.561,23.317,-52.389,179.783,6.815,149.320
C06086=1117.565,23.067,-52.374,179.782,6.810,149.319
C06087=1117.570,22.818,-52.359,179.781,6.806,149.318
C06088=1117.576,22.568,-52.345,179.781,6.801,149.317
C06089=1117.580,22.319,-52.330,179.780,6.797,149.317
C06090=1117.585,22.069,-52.315,179.779,6.793,149.316
C06091=1117.590,21.854,-52.302,179.778,6.789,149.315
C06092=1117.595,21.639,-52.289,179.777,6.785,149.315
C06093=1117.598,21.425,-52.276,179.777,6.781,149.314
C06094=1117.603,21.211,-52.264,179.776,6.778,149.314
C06095=1117.607,20.996,-52.251,179.775,6.773,149.313
C06096=1117.612,20.781,-52.238,179.775,6.770,149.312
C06097=1117.616,20.567,-52.226,179.774,6.766,149.312
C06098=1117.620,20.352,-52.213,179.773,6.762,149.311
C06099=1117.625,20.102,-52.198,179.772,6.758,149.310
C06100=1117.631,19.853,-52.183,179.771,6.753,149.310
C06101=1117.636,19.603,-52.169,179.771,6.749,149.309
C06102=1117.640,19.354,-52.154,179.770,6.744,149.308
C06103=1117.645,19.104,-52.139,179.769,6.740,149.307
C06104=1117.651,18.854,-52.124,179.768,6.735,149.307
C06105=1117.656,18.605,-52.109,179.768,6.732,149.306
C06106=1117.660,18.355,-52.095,179.767,6.727,149.305
C06107=1117.665,18.106,-52.081,179.766,6.723,149.304
C06108=1117.671,17.856,-52.065,179.765,6.718,149.303
C06109=1117.676,17.607,-52.051,179.764,6.714,149.303
C06110=1117.681,17.358,-52.036,179.764,6.709,149.302
C06111=1117.686,17.109,-52.022,179.763,6.705,149.301
C06112=1117.691,16.859,-52.008,179.762,6.700,149.300
C06113=1117.697,16.609,-51.993,179.761,6.696,149.300
C06114=1117.701,16.360,-51.978,179.761,6.691,149.299
C06115=1117.706,16.110,-51.964,179.760,6.687,149.298
C06116=1117.711,15.860,-51.949,179.759,6.682,149.297
C06117=1117.716,15.611,-51.934,179.758,6.678,149.297
C06118=1117.721,15.361,-51.920,179.757,6.673,149.296
C06119=1117.726,15.111,-51.905,179.756,6.669,149.295
C06120=1117.731,14.862,-51.891,179.756,6.664,149.294
C06121=1117.737,14.613,-51.876,179.755,6.659,149.293
C06122=1117.742,14.364,-51.862,179.754,6.655,149.293
C06123=1117.747,14.114,-51.848,179.754,6.650,149.292
C06124=1117.752,13.864,-51.834,179.753,6.646,149.291
C06125=1117.757,13.614,-51.819,179.752,6.641,149.290
C06126=1117.761,13.365,-51.804,179.752,6.636,149.289
C06127=1117.767,13.115,-51.789,179.751,6.632,149.289
C06128=1117.772,12.866,-51.776,179.750,6.627,149.288
C06129=1117.777,12.617,-51.761,179.749,6.623,149.287
C06130=1117.782,12.367,-51.747,179.748,6.618,149.286
C06131=1117.787,12.117,-51.733,179.748,6.614,149.285
C06132=1117.792,11.868,-51.718,179.747,6.609,149.285
C06133=1117.797,11.618,-51.703,179.746,6.605,149.284
C06134=1117.802,11.369,-51.690,179.746,6.600,149.283
C06135=1117.807,11.120,-51.675,179.745,6.595,149.282
C06136=1117.812,10.870,-51.661,179.744,6.591,149.282
C06137=1117.817,10.620,-51.647,179.744,6.586,149.281
C06138=1117.822,10.371,-51.632,179.743,6.581,149.280
C06139=1117.827,10.121,-51.618,179.742,6.577,149.279
C06140=1117.833,9.872,-51.604,179.741,6.572,149.278
C06141=1117.838,9.622,-51.590,179.741,6.568,149.277
C06142=1117.843,9.372,-51.576,179.740,6.563,149.276
C06143=1117.848,9.123,-51.561,179.739,6.559,149.276
C06144=1117.853,8.874,-51.547,179.739,6.554,149.275
C06145=1117.858,8.624,-51.533,179.738,6.549,149.274
C06146=1117.863,8.374,-51.519,179.738,6.544,149.273
C06147=1117.867,8.160,-51.507,179.737,6.541,149.272
C06148=1117.872,7.945,-51.495,179.737,6.537,149.272
C06149=1117.876,7.730,-51.482,179.736,6.533,149.271
C06150=1117.881,7.515,-51.471,179.736,6.529,149.270
C06151=1117.885,7.300,-51.458,179.736,6.526,149.270
C06152=1117.890,7.086,-51.446,179.735,6.521,149.269
C06153=1117.894,6.871,-51.434,179.735,6.517,149.268
C06154=1117.898,6.656,-51.421,179.734,6.514,149.267
C06155=1117.903,6.407,-51.408,179.734,6.509,149.267
C06156=1117.908,6.157,-51.394,179.733,6.504,149.266
C06157=1117.913,5.907,-51.380,179.733,6.500,149.265
C06158=1117.918,5.657,-51.365,179.732,6.495,149.264
C06159=1117.924,5.408,-51.352,179.732,6.491,149.263
C06160=1117.929,5.159,-51.337,179.731,6.487,149.262
C06161=1117.934,4.909,-51.323,179.731,6.482,149.261
C06162=1117.939,4.660,-51.310,179.730,6.477,149.261
C06163=1117.944,4.411,-51.295,179.729,6.473,149.260
C06164=1117.949,4.160,-51.282,179.729,6.468,149.259
C06165=1117.954,3.911,-51.268,179.728,6.463,149.258
C06166=1117.959,3.661,-51.254,179.727,6.459,149.257
C06167=1117.964,3.412,-51.239,179.727,6.455,149.256
C06168=1117.969,3.163,-51.226,179.727,6.450,149.255
C06169=1117.974,2.913,-51.212,179.726,6.445,149.255
C06170=1117.979,2.663,-51.198,179.725,6.441,149.254
C06171=1117.985,2.414,-51.184,179.725,6.436,149.253
C06172=1117.990,2.164,-51.170,179.724,6.432,149.252
C06173=1117.994,1.914,-51.157,179.724,6.427,149.251
C06174=1118.000,1.665,-51.143,179.723,6.423,149.251
C06175=1118.005,1.416,-51.129,179.723,6.419,149.250
C06176=1118.010,1.166,-51.115,179.722,6.414,149.249
C06177=1118.016,0.916,-51.101,179.722,6.409,149.248
C06178=1118.020,0.667,-51.088,179.721,6.405,149.247
C06179=1118.025,0.417,-51.073,179.720,6.400,149.246
C06180=1118.031,0.167,-51.060,179.720,6.395,149.246
C06181=1118.036,-0.082,-51.046,179.719,6.391,149.245
C06182=1118.040,-0.331,-51.033,179.719,6.387,149.244
C06183=1118.046,-0.581,-51.019,179.718,6.382,149.243
C06184=1118.051,-0.831,-51.005,179.718,6.378,149.242
C06185=1118.056,-1.080,-50.991,179.717,6.373,149.241
C06186=1118.061,-1.330,-50.978,179.716,6.369,149.241
C06187=1118.066,-1.579,-50.964,179.716,6.364,149.240
C06188=1118.072,-1.829,-50.950,179.715,6.359,149.239
C06189=1118.076,-2.079,-50.937,179.714,6.355,149.238
C06190=1118.081,-2.328,-50.923,179.714,6.350,149.237
C06191=1118.087,-2.578,-50.909,179.714,6.346,149.236
C06192=1118.091,-2.827,-50.896,179.713,6.342,149.236
C06193=1118.097,-3.077,-50.882,179.712,6.337,149.235
C06194=1118.102,-3.326,-50.868,179.712,6.333,149.234
C06195=1118.107,-3.576,-50.856,179.711,6.328,149.233
C06196=1118.112,-3.826,-50.841,179.710,6.323,149.232
C06197=1118.118,-4.075,-50.828,179.710,6.319,149.232
C06198=1118.122,-4.325,-50.814,179.709,6.314,149.231
C06199=1118.128,-4.574,-50.801,179.709,6.309,149.230
C06200=1118.133,-4.824,-50.787,179.708,6.306,149.229
C06201=1118.138,-5.074,-50.774,179.708,6.301,149.228
C06202=1118.143,-5.323,-50.760,179.707,6.296,149.227
C06203=1118.147,-5.538,-50.749,179.706,6.292,149.227
C06204=1118.152,-5.753,-50.737,179.706,6.288,149.226
C06205=1118.156,-5.968,-50.726,179.705,6.285,149.225
C06206=1118.161,-6.183,-50.714,179.704,6.281,149.225
C06207=1118.165,-6.398,-50.702,179.705,6.277,149.224
C06208=1118.170,-6.613,-50.691,179.704,6.273,149.223
C06209=1118.173,-6.827,-50.679,179.703,6.269,149.222
C06210=1118.178,-7.042,-50.667,179.703,6.265,149.222
C06211=1118.183,-7.292,-50.654,179.702,6.260,149.221
C06212=1118.189,-7.542,-50.641,179.701,6.256,149.220
C06213=1118.193,-7.791,-50.627,179.701,6.251,149.219
C06214=1118.199,-8.041,-50.614,179.700,6.247,149.218
C06215=1118.203,-8.289,-50.601,179.700,6.242,149.218
C06216=1118.209,-8.540,-50.587,179.699,6.238,149.217
C06217=1118.214,-8.789,-50.575,179.698,6.233,149.216
C06218=1118.219,-9.039,-50.561,179.698,6.228,149.215
C06219=1118.224,-9.288,-50.548,179.697,6.224,149.214
C06220=1118.229,-9.538,-50.534,179.697,6.220,149.214
C06221=1118.234,-9.788,-50.522,179.696,6.215,149.213
C06222=1118.239,-10.037,-50.507,179.695,6.211,149.212
C06223=1118.244,-10.287,-50.495,179.695,6.206,149.211
C06224=1118.250,-10.537,-50.481,179.694,6.201,149.210
C06225=1118.254,-10.786,-50.468,179.693,6.197,149.210
C06226=1118.260,-11.035,-50.455,179.693,6.192,149.209
C06227=1118.265,-11.285,-50.442,179.692,6.188,149.208
C06228=1118.270,-11.535,-50.429,179.692,6.183,149.207
C06229=1118.275,-11.784,-50.415,179.691,6.179,149.206
C06230=1118.280,-12.034,-50.402,179.690,6.174,149.205
C06231=1118.286,-12.283,-50.389,179.690,6.169,149.204
C06232=1118.290,-12.533,-50.376,179.689,6.165,149.204
C06233=1118.296,-12.783,-50.363,179.688,6.160,149.203
C06234=1118.301,-13.032,-50.349,179.688,6.155,149.202
C06235=1118.306,-13.282,-50.337,179.687,6.151,149.201
C06236=1118.312,-13.531,-50.324,179.686,6.146,149.200
C06237=1118.316,-13.781,-50.311,179.686,6.141,149.200
C06238=1118.321,-14.031,-50.298,179.685,6.137,149.199
C06239=1118.326,-14.281,-50.284,179.685,6.132,149.198
C06240=1118.332,-14.530,-50.272,179.684,6.128,149.197
C06241=1118.337,-14.780,-50.259,179.683,6.123,149.196
C06242=1118.342,-15.029,-50.245,179.683,6.118,149.195
C06243=1118.347,-15.279,-50.232,179.682,6.114,149.194
C06244=1118.353,-15.528,-50.219,179.681,6.109,149.194
C06245=1118.357,-15.778,-50.206,179.681,6.104,149.193
C06246=1118.362,-16.028,-50.194,179.680,6.100,149.192
C06247=1118.368,-16.277,-50.180,179.680,6.095,149.191
C06248=1118.373,-16.527,-50.167,179.679,6.091,149.190
C06249=1118.378,-16.777,-50.155,179.678,6.086,149.190
C06250=1118.383,-17.026,-50.142,179.678,6.081,149.189
C06251=1118.388,-17.276,-50.129,179.677,6.076,149.188
C06252=1118.393,-17.525,-50.116,179.677,6.072,149.187
C06253=1118.398,-17.775,-50.103,179.676,6.067,149.186
C06254=1118.404,-18.024,-50.091,179.676,6.063,149.185
C06255=1118.409,-18.274,-50.077,179.675,6.058,149.184
C06256=1118.414,-18.524,-50.065,179.675,6.053,149.183
C06257=1118.419,-18.773,-50.052,179.674,6.049,149.183
C06258=1118.424,-19.023,-50.039,179.673,6.044,149.182
C06259=1118.429,-19.238,-50.028,179.673,6.039,149.181
C06260=1118.433,-19.453,-50.017,179.672,6.036,149.180
C06261=1118.438,-19.668,-50.005,179.671,6.031,149.180
C06262=1118.442,-19.883,-49.995,179.671,6.028,149.179
C06263=1118.447,-20.098,-49.984,179.670,6.023,149.178
C06264=1118.451,-20.313,-49.973,179.670,6.020,149.177
C06265=1118.455,-20.528,-49.962,179.669,6.015,149.177
C06266=1118.460,-20.742,-49.951,179.669,6.011,149.176
C06267=1118.464,-20.992,-49.938,179.668,6.006,149.175
C06268=1118.470,-21.242,-49.926,179.667,6.001,149.174
C06269=1118.476,-21.492,-49.913,179.667,5.997,149.173
C06270=1118.481,-21.741,-49.901,179.666,5.992,149.173
C06271=1118.485,-21.991,-49.888,179.666,5.987,149.172
C06272=1118.491,-22.240,-49.875,179.665,5.983,149.171
C06273=1118.496,-22.490,-49.863,179.665,5.978,149.170
C06274=1118.501,-22.740,-49.850,179.664,5.973,149.169
C06275=1118.506,-22.989,-49.838,179.663,5.968,149.168
C06276=1118.511,-23.239,-49.824,179.663,5.963,149.167
C06277=1118.517,-23.489,-49.812,179.662,5.958,149.166
C06278=1118.522,-23.739,-49.800,179.661,5.954,149.166
C06279=1118.527,-23.988,-49.787,179.661,5.949,149.165
C06280=1118.532,-24.237,-49.775,179.660,5.944,149.164
C06281=1118.537,-24.487,-49.762,179.660,5.940,149.163
C06282=1118.542,-24.737,-49.750,179.659,5.934,149.162
C06283=1118.547,-24.987,-49.737,179.658,5.929,149.161
C06284=1118.552,-25.236,-49.725,179.658,5.925,149.160
C06285=1118.558,-25.486,-49.713,179.657,5.920,149.159
C06286=1118.563,-25.735,-49.700,179.657,5.915,149.158
C06287=1118.568,-25.984,-49.687,179.657,5.910,149.157
C06288=1118.574,-26.234,-49.676,179.657,5.906,149.156
C06289=1118.578,-26.484,-49.663,179.658,5.902,149.155
C06290=1118.583,-26.734,-49.650,179.658,5.897,149.154
C06291=1118.589,-26.984,-49.638,179.659,5.894,149.153
C06292=1118.595,-27.233,-49.625,179.660,5.890,149.152
C06293=1118.600,-27.483,-49.612,179.660,5.886,149.151
C06294=1118.605,-27.732,-49.600,179.661,5.881,149.150
C06295=1118.610,-27.982,-49.588,179.661,5.877,149.149
C06296=1118.615,-28.232,-49.576,179.661,5.872,149.148
C06297=1118.620,-28.482,-49.563,179.661,5.868,149.147
C06298=1118.625,-28.731,-49.550,179.662,5.864,149.146
C06299=1118.631,-28.981,-49.539,179.662,5.860,149.145
C06300=1118.635,-29.230,-49.527,179.662,5.856,149.144
C06301=1118.641,-29.480,-49.515,179.663,5.852,149.143
C06302=1118.646,-29.729,-49.502,179.662,5.847,149.142
C06303=1118.651,-29.979,-49.489,179.662,5.843,149.141
C06304=1118.656,-30.229,-49.478,179.663,5.839,149.140
C06305=1118.661,-30.478,-49.465,179.663,5.835,149.139
C06306=1118.666,-30.728,-49.453,179.663,5.830,149.138
C06307=1118.671,-30.978,-49.440,179.663,5.826,149.137
C06308=1118.677,-31.228,-49.428,179.662,5.821,149.136
C06309=1118.682,-31.477,-49.416,179.662,5.817,149.135
C06310=1118.687,-31.727,-49.404,179.663,5.813,149.134
C06311=1118.692,-31.976,-49.391,179.662,5.809,149.134
C06312=1118.698,-32.226,-49.379,179.662,5.804,149.133
C06313=1118.703,-32.476,-49.367,179.662,5.800,149.132
C06314=1118.708,-32.726,-49.355,179.661,5.795,149.131
C06315=1118.712,-32.940,-49.344,179.662,5.791,149.130
C06316=1118.717,-33.156,-49.333,179.661,5.788,149.129
C06317=1118.721,-33.370,-49.323,179.661,5.784,149.129
C06318=1118.726,-33.585,-49.313,179.661,5.780,149.128
C06319=1118.731,-33.801,-49.302,179.660,5.776,149.127
C06320=1118.735,-34.015,-49.292,179.660,5.772,149.126
C06321=1118.739,-34.231,-49.281,179.659,5.769,149.126
C06322=1118.743,-34.446,-49.271,179.660,5.765,149.125
C06323=1118.749,-34.695,-49.259,179.659,5.761,149.124
C06324=1118.754,-34.945,-49.246,179.658,5.756,149.123
C06325=1118.759,-35.195,-49.234,179.658,5.751,149.122
C06326=1118.765,-35.445,-49.222,179.657,5.746,149.121
C06327=1118.769,-35.694,-49.210,179.656,5.742,149.121
C06328=1118.775,-35.944,-49.199,179.656,5.737,149.120
C06329=1118.780,-36.193,-49.186,179.655,5.732,149.119
C06330=1118.785,-36.443,-49.174,179.654,5.728,149.118
C06331=1118.791,-36.693,-49.162,179.653,5.723,149.117
C06332=1118.796,-36.942,-49.150,179.653,5.718,149.116
C06333=1118.800,-37.192,-49.138,179.652,5.713,149.116
C06334=1118.806,-37.442,-49.126,179.652,5.709,149.115
C06335=1118.811,-37.691,-49.114,179.650,5.704,149.114
C06336=1118.816,-37.941,-49.102,179.650,5.699,149.113
C06337=1118.821,-38.191,-49.091,179.649,5.694,149.112
C06338=1118.827,-38.441,-49.079,179.648,5.689,149.112
C06339=1118.832,-38.690,-49.066,179.647,5.684,149.111
C06340=1118.838,-38.939,-49.055,179.646,5.679,149.110
C06341=1118.842,-39.189,-49.043,179.645,5.674,149.109
C06342=1118.848,-39.439,-49.031,179.644,5.669,149.108
C06343=1118.853,-39.689,-49.020,179.643,5.664,149.108
C06344=1118.858,-39.938,-49.007,179.642,5.659,149.107
C06345=1118.863,-40.187,-48.996,179.641,5.654,149.106
C06346=1118.869,-40.437,-48.984,179.640,5.648,149.105
C06347=1118.874,-40.687,-48.972,179.638,5.643,149.104
C06348=1118.879,-40.937,-48.961,179.637,5.637,149.104
C06349=1118.884,-41.187,-48.949,179.636,5.632,149.103
C06350=1118.889,-41.436,-48.936,179.635,5.628,149.102
C06351=1118.895,-41.685,-48.925,179.634,5.622,149.101
C06352=1118.900,-41.935,-48.913,179.632,5.616,149.100
C06353=1118.905,-42.185,-48.901,179.631,5.610,149.100
C06354=1118.910,-42.435,-48.890,179.629,5.605,149.099
C06355=1118.916,-42.685,-48.878,179.628,5.600,149.098
C06356=1118.920,-42.934,-48.867,179.627,5.594,149.097
C06357=1118.926,-43.184,-48.855,179.627,5.589,149.096
C06358=1118.932,-43.433,-48.844,179.627,5.584,149.095
C06359=1118.936,-43.683,-48.832,179.628,5.580,149.094
C06360=1118.942,-43.933,-48.820,179.627,5.575,149.093
C06361=1118.946,-44.183,-48.809,179.627,5.570,149.092
C06362=1118.952,-44.433,-48.797,179.628,5.566,149.091
C06363=1118.958,-44.682,-48.786,179.627,5.561,149.090
C06364=1118.963,-44.931,-48.774,179.628,5.557,149.089
C06365=1118.968,-45.181,-48.763,179.628,5.552,149.087
C06366=1118.973,-45.431,-48.751,179.628,5.546,149.086
C06367=1118.978,-45.681,-48.739,179.628,5.542,149.085
C06368=1118.983,-45.930,-48.728,179.628,5.537,149.084
C06369=1118.989,-46.180,-48.717,179.629,5.533,149.083
C06370=1118.994,-46.429,-48.705,179.629,5.528,149.082
C06371=1118.998,-46.644,-48.695,179.629,5.524,149.081
C06372=1119.003,-46.860,-48.685,179.630,5.520,149.080
C06373=1119.008,-47.075,-48.675,179.630,5.516,149.079
C06374=1119.012,-47.290,-48.665,179.630,5.512,149.078
C06375=1119.017,-47.505,-48.656,179.630,5.508,149.077
C06376=1119.021,-47.720,-48.646,179.630,5.503,149.076
C06377=1119.025,-47.935,-48.636,179.630,5.499,149.076
C06378=1119.030,-48.150,-48.627,179.630,5.495,149.075
C06379=1119.035,-48.400,-48.615,179.631,5.491,149.074
C06380=1119.040,-48.650,-48.604,179.631,5.486,149.072
C06381=1119.046,-48.900,-48.592,179.630,5.481,149.071
C06382=1119.051,-49.149,-48.581,179.631,5.477,149.070
C06383=1119.056,-49.399,-48.569,179.631,5.472,149.069
C06384=1119.061,-49.649,-48.558,179.631,5.468,149.068
C06385=1119.067,-49.899,-48.546,179.631,5.463,149.067
C06386=1119.072,-50.148,-48.536,179.631,5.458,149.066
C06387=1119.077,-50.398,-48.524,179.632,5.454,149.065
C06388=1119.082,-50.648,-48.512,179.632,5.448,149.064
C06389=1119.088,-50.897,-48.502,179.632,5.444,149.063
C06390=1119.093,-51.147,-48.490,179.632,5.439,149.062
C06391=1119.098,-51.397,-48.479,179.632,5.434,149.061
C06392=1119.103,-51.647,-48.467,179.633,5.430,149.060
C06393=1119.109,-51.895,-48.456,179.633,5.425,149.058
C06394=1119.114,-52.146,-48.446,179.633,5.421,149.057
C06395=1119.119,-52.396,-48.434,179.633,5.416,149.056
C06396=1119.124,-52.645,-48.423,179.634,5.411,149.055
C06397=1119.130,-52.895,-48.411,179.633,5.407,149.054
C06398=1119.135,-53.145,-48.400,179.633,5.401,149.053
C06399=1119.140,-53.394,-48.389,179.634,5.397,149.052
C06400=1119.145,-53.644,-48.378,179.634,5.392,149.051
C06401=1119.150,-53.893,-48.366,179.634,5.388,149.050
C06402=1119.155,-54.144,-48.356,179.634,5.383,149.049
C06403=1119.161,-54.393,-48.344,179.634,5.378,149.048
C06404=1119.166,-54.642,-48.333,179.635,5.374,149.047
C06405=1119.171,-54.893,-48.322,179.635,5.369,149.046
C06406=1119.177,-55.142,-48.311,179.635,5.365,149.045
C06407=1119.182,-55.391,-48.299,179.635,5.360,149.043
C06408=1119.187,-55.642,-48.289,179.635,5.354,149.042
C06409=1119.193,-55.891,-48.277,179.635,5.350,149.041
C06410=1119.197,-56.141,-48.266,179.635,5.345,149.040
C06411=1119.202,-56.391,-48.256,179.636,5.341,149.039
C06412=1119.208,-56.640,-48.244,179.636,5.336,149.038
C06413=1119.213,-56.890,-48.233,179.636,5.331,149.037
C06414=1119.219,-57.139,-48.222,179.637,5.327,149.036
C06415=1119.223,-57.389,-48.211,179.636,5.322,149.035
C06416=1119.229,-57.639,-48.200,179.637,5.318,149.034
C06417=1119.234,-57.888,-48.189,179.636,5.313,149.033
C06418=1119.239,-58.139,-48.179,179.637,5.309,149.032
C06419=1119.244,-58.388,-48.167,179.637,5.303,149.031
C06420=1119.250,-58.637,-48.156,179.637,5.299,149.030
C06421=1119.255,-58.888,-48.145,179.637,5.294,149.028
C06422=1119.260,-59.137,-48.134,179.638,5.289,149.027
C06423=1119.265,-59.387,-48.124,179.638,5.285,149.026
C06424=1119.271,-59.637,-48.112,179.638,5.280,149.025
C06425=1119.276,-59.886,-48.102,179.638,5.275,149.024
C06426=1119.281,-60.136,-48.090,179.638,5.271,149.023
C06427=1119.286,-60.351,-48.081,179.637,5.267,149.022
C06428=1119.290,-60.566,-48.071,179.637,5.262,149.022
C06429=1119.295,-60.782,-48.062,179.636,5.257,149.021
C06430=1119.299,-60.997,-48.052,179.636,5.253,149.020
C06431=1119.305,-61.212,-48.043,179.635,5.248,149.019
C06432=1119.308,-61.427,-48.034,179.635,5.244,149.018
C06433=1119.313,-61.642,-48.025,179.634,5.240,149.018
C06434=1119.317,-61.858,-48.015,179.634,5.235,149.017
C06435=1119.322,-62.107,-48.004,179.633,5.230,149.016
C06436=1119.328,-62.357,-47.994,179.632,5.225,149.015
C06437=1119.333,-62.607,-47.983,179.631,5.219,149.014
C06438=1119.339,-62.856,-47.972,179.631,5.215,149.013
C06439=1119.344,-63.107,-47.961,179.630,5.209,149.012
C06440=1119.349,-63.355,-47.950,179.630,5.204,149.011
C06441=1119.354,-63.606,-47.940,179.629,5.198,149.010
C06442=1119.360,-63.855,-47.930,179.629,5.194,149.009
C06443=1119.364,-64.105,-47.918,179.628,5.188,149.008
C06444=1119.370,-64.354,-47.908,179.627,5.183,149.007
C06445=1119.376,-64.605,-47.897,179.627,5.178,149.006
C06446=1119.381,-64.854,-47.886,179.626,5.173,149.005
C06447=1119.386,-65.104,-47.875,179.626,5.168,149.004
C06448=1119.392,-65.354,-47.865,179.626,5.162,149.003
C06449=1119.396,-65.603,-47.854,179.625,5.157,149.002
C06450=1119.402,-65.853,-47.844,179.624,5.152,149.001
C06451=1119.407,-66.103,-47.833,179.624,5.146,149.000
C06452=1119.412,-66.353,-47.823,179.624,5.142,148.999
C06453=1119.417,-66.602,-47.812,179.624,5.136,148.998
C06454=1119.423,-66.852,-47.801,179.623,5.131,148.997
C06455=1119.428,-67.102,-47.791,179.622,5.125,148.996
C06456=1119.433,-67.352,-47.781,179.622,5.120,148.995
C06457=1119.438,-67.601,-47.769,179.622,5.115,148.994
C06458=1119.444,-67.851,-47.759,179.621,5.109,148.993
C06459=1119.449,-68.100,-47.749,179.621,5.105,148.992
C06460=1119.454,-68.351,-47.738,179.621,5.100,148.991
C06461=1119.460,-68.600,-47.728,179.620,5.094,148.990
C06462=1119.464,-68.850,-47.717,179.620,5.089,148.989
C06463=1119.470,-69.099,-47.707,179.620,5.084,148.988
C06464=1119.476,-69.349,-47.696,179.620,5.078,148.987
C06465=1119.481,-69.599,-47.686,179.619,5.073,148.986
C06466=1119.486,-69.849,-47.676,179.619,5.068,148.985
C06467=1119.491,-70.099,-47.665,179.619,5.062,148.984
C06468=1119.497,-70.348,-47.655,179.619,5.058,148.983
C06469=1119.502,-70.598,-47.645,179.619,5.052,148.981
C06470=1119.507,-70.848,-47.634,179.618,5.046,148.980
C06471=1119.513,-71.097,-47.623,179.618,5.042,148.979
C06472=1119.518,-71.346,-47.614,179.618,5.036,148.978
C06473=1119.523,-71.597,-47.603,179.617,5.031,148.977
C06474=1119.528,-71.846,-47.593,179.617,5.026,148.976
C06475=1119.533,-72.096,-47.582,179.617,5.021,148.975
C06476=1119.539,-72.346,-47.572,179.617,5.015,148.974
C06477=1119.544,-72.595,-47.562,179.616,5.010,148.973
C06478=1119.549,-72.846,-47.551,179.617,5.005,148.972
C06479=1119.555,-73.095,-47.541,179.617,5.000,148.971
C06480=1119.560,-73.344,-47.531,179.617,4.994,148.969
C06481=1119.565,-73.595,-47.521,179.617,4.990,148.968
C06482=1119.570,-73.844,-47.511,179.616,4.984,148.967
C06483=1119.575,-74.060,-47.501,179.616,4.980,148.966
C06484=1119.580,-74.275,-47.494,179.616,4.975,148.965
C06485=1119.585,-74.490,-47.484,179.617,4.971,148.964
C06486=1119.589,-74.706,-47.475,179.616,4.966,148.963
C06487=1119.594,-74.920,-47.467,179.616,4.961,148.962
C06488=1119.599,-75.136,-47.458,179.616,4.957,148.961
C06489=1119.603,-75.352,-47.450,179.616,4.952,148.961
C06490=1119.607,-75.567,-47.440,179.616,4.948,148.960
C06491=1119.613,-75.817,-47.430,179.616,4.943,148.958
C06492=1119.618,-76.066,-47.420,179.616,4.937,148.957
C06493=1119.623,-76.315,-47.410,179.616,4.932,148.956
C06494=1119.629,-76.566,-47.400,179.616,4.927,148.955
C06495=1119.634,-76.816,-47.390,179.616,4.922,148.954
C06496=1119.640,-77.065,-47.380,179.616,4.917,148.953
C06497=1119.645,-77.315,-47.370,179.617,4.912,148.951
C06498=1119.650,-77.565,-47.360,179.617,4.906,148.950
C06499=1119.655,-77.814,-47.350,179.617,4.901,148.949
C06500=1119.661,-78.065,-47.340,179.617,4.896,148.948
C06501=1119.666,-78.314,-47.330,179.617,4.891,148.947
C06502=1119.671,-78.564,-47.320,179.617,4.886,148.946
C06503=1119.677,-78.814,-47.310,179.617,4.881,148.945
C06504=1119.681,-79.063,-47.300,179.617,4.875,148.944
C06505=1119.687,-79.313,-47.291,179.617,4.870,148.942
C06506=1119.693,-79.562,-47.280,179.617,4.865,148.941
C06507=1119.698,-79.813,-47.270,179.617,4.860,148.940
C06508=1119.703,-80.062,-47.260,179.618,4.854,148.939
C06509=1119.709,-80.312,-47.251,179.618,4.849,148.937
C06510=1119.714,-80.562,-47.240,179.619,4.845,148.936
C06511=1119.719,-80.811,-47.231,179.619,4.839,148.935
C06512=1119.724,-81.061,-47.220,179.619,4.834,148.934
C06513=1119.730,-81.311,-47.211,179.619,4.829,148.933
C06514=1119.735,-81.561,-47.201,179.619,4.824,148.932
C06515=1119.741,-81.810,-47.191,179.619,4.819,148.930
C06516=1119.746,-82.060,-47.181,179.620,4.814,148.929
C06517=1119.751,-82.310,-47.171,179.620,4.808,148.928
C06518=1119.756,-82.560,-47.161,179.620,4.803,148.927
C06519=1119.761,-82.810,-47.152,179.620,4.798,148.926
C06520=1119.767,-83.059,-47.142,179.620,4.793,148.925
C06521=1119.773,-83.309,-47.132,179.620,4.788,148.923
C06522=1119.778,-83.558,-47.123,179.621,4.783,148.922
C06523=1119.783,-83.808,-47.113,179.622,4.778,148.921
C06524=1119.788,-84.058,-47.103,179.622,4.773,148.920
C06525=1119.794,-84.308,-47.093,179.622,4.768,148.918
C06526=1119.799,-84.558,-47.083,179.622,4.762,148.917
C06527=1119.804,-84.808,-47.074,179.623,4.757,148.916
C06528=1119.810,-85.057,-47.064,179.623,4.753,148.915
C06529=1119.815,-85.306,-47.054,179.624,4.748,148.914
C06530=1119.821,-85.556,-47.045,179.624,4.743,148.913
C06531=1119.825,-85.806,-47.035,179.624,4.737,148.911
C06532=1119.831,-86.057,-47.025,179.625,4.733,148.910
C06533=1119.836,-86.306,-47.016,179.625,4.728,148.909
C06534=1119.842,-86.556,-47.006,179.626,4.722,148.908
C06535=1119.847,-86.805,-46.996,179.626,4.717,148.906
C06536=1119.852,-87.055,-46.987,179.626,4.713,148.905
C06537=1119.858,-87.305,-46.977,179.627,4.707,148.904
C06538=1119.863,-87.554,-46.967,179.627,4.702,148.903
C06539=1119.867,-87.770,-46.959,179.628,4.698,148.902
C06540=1119.872,-87.986,-46.951,179.628,4.694,148.901
C06541=1119.877,-88.200,-46.943,179.629,4.690,148.900
C06542=1119.881,-88.416,-46.935,179.629,4.686,148.898
C06543=1119.886,-88.632,-46.926,179.630,4.682,148.897
C06544=1119.890,-88.847,-46.918,179.630,4.676,148.896
C06545=1119.895,-89.062,-46.910,179.630,4.672,148.895
C06546=1119.900,-89.278,-46.901,179.631,4.668,148.894
C06547=1119.905,-89.527,-46.892,179.632,4.664,148.893
C06548=1119.911,-89.777,-46.882,179.632,4.659,148.892
C06549=1119.916,-90.027,-46.873,179.632,4.653,148.891
C06550=1119.921,-90.277,-46.864,179.633,4.649,148.889
C06551=1119.926,-90.526,-46.854,179.633,4.644,148.888
C06552=1119.932,-90.776,-46.845,179.634,4.639,148.887
C06553=1119.937,-91.026,-46.835,179.635,4.634,148.886
C06554=1119.942,-91.276,-46.825,179.635,4.630,148.884
C06555=1119.948,-91.526,-46.816,179.636,4.625,148.883
C06556=1119.952,-91.775,-46.806,179.636,4.620,148.882
C06557=1119.958,-92.026,-46.797,179.637,4.615,148.881
C06558=1119.963,-92.275,-46.787,179.638,4.610,148.879
C06559=1119.968,-92.525,-46.778,179.638,4.605,148.878
C06560=1119.974,-92.775,-46.769,179.639,4.601,148.877
C06561=1119.979,-93.024,-46.759,179.640,4.595,148.876
C06562=1119.985,-93.274,-46.750,179.640,4.591,148.874
C06563=1119.990,-93.524,-46.741,179.641,4.587,148.873
C06564=1119.995,-93.773,-46.731,179.641,4.581,148.872
C06565=1120.001,-94.024,-46.722,179.642,4.577,148.871
C06566=1120.006,-94.273,-46.713,179.643,4.572,148.869
C06567=1120.012,-94.523,-46.702,179.644,4.567,148.868
C06568=1120.017,-94.773,-46.694,179.644,4.562,148.867
C06569=1120.022,-95.023,-46.685,179.644,4.558,148.866
C06570=1120.028,-95.272,-46.674,179.644,4.553,148.865
C06571=1120.033,-95.522,-46.666,179.644,4.548,148.864
C06572=1120.038,-95.772,-46.657,179.645,4.543,148.863
C06573=1120.044,-96.021,-46.646,179.645,4.538,148.861
C06574=1120.049,-96.271,-46.638,179.646,4.533,148.860
C06575=1120.054,-96.521,-46.629,179.646,4.528,148.859
C06576=1120.060,-96.771,-46.619,179.646,4.523,148.858
C06577=1120.065,-97.020,-46.610,179.646,4.518,148.857
C06578=1120.070,-97.270,-46.601,179.647,4.513,148.855
C06579=1120.076,-97.521,-46.591,179.647,4.508,148.854
C06580=1120.081,-97.770,-46.582,179.648,4.503,148.853
C06581=1120.086,-98.019,-46.573,179.648,4.498,148.852
C06582=1120.092,-98.269,-46.564,179.649,4.493,148.851
C06583=1120.098,-98.519,-46.555,179.649,4.488,148.850
C06584=1120.103,-98.769,-46.546,179.648,4.483,148.849
C06585=1120.109,-99.019,-46.536,179.649,4.478,148.847
C06586=1120.113,-99.268,-46.527,179.649,4.473,148.846
C06587=1120.119,-99.518,-46.518,179.650,4.469,148.845
C06588=1120.124,-99.768,-46.509,179.650,4.464,148.844
C06589=1120.130,-100.018,-46.499,179.650,4.458,148.843
C06590=1120.135,-100.268,-46.490,179.650,4.453,148.841
C06591=1120.140,-100.517,-46.481,179.651,4.448,148.840
C06592=1120.145,-100.767,-46.472,179.651,4.444,148.839
C06593=1120.151,-101.017,-46.462,179.652,4.439,148.838
C06594=1120.157,-101.266,-46.454,179.652,4.433,148.837
C06595=1120.161,-101.482,-46.446,179.652,4.429,148.836
C06596=1120.166,-101.697,-46.438,179.652,4.425,148.835
C06597=1120.170,-101.913,-46.430,179.653,4.420,148.834
C06598=1120.175,-102.128,-46.423,179.653,4.416,148.833
C06599=1120.179,-102.344,-46.415,179.653,4.411,148.832
C06600=1120.184,-102.559,-46.407,179.653,4.408,148.831
C06601=1120.189,-102.775,-46.399,179.654,4.403,148.830
C06602=1120.193,-102.990,-46.391,179.654,4.398,148.829
C06603=1120.199,-103.240,-46.382,179.654,4.393,148.827
C06604=1120.204,-103.490,-46.373,179.655,4.389,148.826
C06605=1120.209,-103.740,-46.364,179.655,4.384,148.825
C06606=1120.214,-103.990,-46.355,179.655,4.379,148.824
C06607=1120.221,-104.239,-46.346,179.655,4.373,148.823
C06608=1120.226,-104.489,-46.337,179.655,4.369,148.822
C06609=1120.231,-104.739,-46.328,179.655,4.363,148.820
C06610=1120.236,-104.989,-46.320,179.655,4.358,148.819
C06611=1120.241,-105.238,-46.311,179.656,4.353,148.818
C06612=1120.246,-105.488,-46.302,179.657,4.349,148.817
C06613=1120.252,-105.738,-46.293,179.657,4.344,148.816
C06614=1120.257,-105.987,-46.284,179.657,4.338,148.814
C06615=1120.263,-106.237,-46.275,179.657,4.333,148.813
C06616=1120.268,-106.487,-46.266,179.657,4.328,148.812
C06617=1120.274,-106.737,-46.257,179.658,4.323,148.811
C06618=1120.279,-106.987,-46.248,179.658,4.318,148.810
C06619=1120.284,-107.237,-46.239,179.658,4.313,148.808
C06620=1120.290,-107.486,-46.231,179.658,4.307,148.807
C06621=1120.295,-107.736,-46.222,179.659,4.302,148.806
C06622=1120.300,-107.986,-46.213,179.659,4.297,148.805
C06623=1120.305,-108.236,-46.205,179.659,4.292,148.804
C06624=1120.311,-108.486,-46.196,179.660,4.288,148.803
C06625=1120.316,-108.735,-46.187,179.660,4.282,148.801
C06626=1120.322,-108.985,-46.178,179.661,4.277,148.800
C06627=1120.327,-109.235,-46.169,179.661,4.272,148.799
C06628=1120.333,-109.485,-46.160,179.661,4.267,148.798
C06629=1120.338,-109.734,-46.151,179.661,4.262,148.797
C06630=1120.344,-109.984,-46.143,179.662,4.257,148.795
C06631=1120.349,-110.235,-46.134,179.662,4.251,148.794
C06632=1120.354,-110.484,-46.125,179.662,4.246,148.793
C06633=1120.360,-110.734,-46.117,179.662,4.241,148.792
C06634=1120.365,-110.983,-46.108,179.663,4.236,148.791
C06635=1120.370,-111.233,-46.099,179.663,4.231,148.789
C06636=1120.375,-111.483,-46.090,179.663,4.226,148.788
C06637=1120.382,-111.733,-46.082,179.663,4.220,148.787
C06638=1120.387,-111.983,-46.074,179.664,4.215,148.786
C06639=1120.392,-112.233,-46.065,179.664,4.210,148.785
C06640=1120.397,-112.482,-46.056,179.664,4.205,148.783
C06641=1120.403,-112.732,-46.048,179.664,4.200,148.782
C06642=1120.408,-112.982,-46.039,179.665,4.194,148.781
C06643=1120.413,-113.232,-46.030,179.665,4.189,148.780
C06644=1120.419,-113.481,-46.022,179.665,4.184,148.779
C06645=1120.425,-113.731,-46.013,179.665,4.179,148.777
C06646=1120.430,-113.981,-46.005,179.666,4.174,148.776
C06647=1120.434,-114.231,-45.996,179.665,4.168,148.775
C06648=1120.440,-114.480,-45.988,179.666,4.163,148.774
C06649=1120.446,-114.730,-45.979,179.666,4.157,148.772
C06650=1120.451,-114.980,-45.971,179.666,4.152,148.771
C06651=1120.456,-115.195,-45.963,179.666,4.148,148.770
C06652=1120.461,-115.411,-45.956,179.666,4.144,148.769
C06653=1120.465,-115.627,-45.948,179.667,4.139,148.768
C06654=1120.470,-115.843,-45.941,179.667,4.134,148.767
C06655=1120.475,-116.058,-45.934,179.667,4.130,148.766
C06656=1120.479,-116.273,-45.927,179.667,4.125,148.765
C06657=1120.483,-116.489,-45.919,179.668,4.121,148.764
C06658=1120.488,-116.705,-45.912,179.668,4.116,148.763
C06659=1120.494,-116.955,-45.904,179.668,4.111,148.762
C06660=1120.500,-117.204,-45.896,179.669,4.106,148.760
C06661=1120.505,-117.454,-45.887,179.669,4.101,148.759
C06662=1120.510,-117.704,-45.878,179.669,4.095,148.758
C06663=1120.515,-117.953,-45.871,179.669,4.089,148.757
C06664=1120.521,-118.203,-45.862,179.669,4.084,148.756
C06665=1120.527,-118.453,-45.854,179.669,4.079,148.754
C06666=1120.532,-118.703,-45.845,179.670,4.074,148.753
C06667=1120.537,-118.953,-45.836,179.670,4.069,148.752
C06668=1120.543,-119.203,-45.828,179.670,4.064,148.751
C06669=1120.547,-119.452,-45.820,179.670,4.058,148.750
C06670=1120.553,-119.703,-45.812,179.671,4.052,148.748
C06671=1120.559,-119.952,-45.803,179.671,4.047,148.747
C06672=1120.564,-120.202,-45.795,179.671,4.042,148.746
C06673=1120.570,-120.451,-45.787,179.671,4.036,148.745
C06674=1120.575,-120.702,-45.779,179.672,4.031,148.743
C06675=1120.580,-120.951,-45.770,179.671,4.025,148.742
C06676=1120.586,-121.201,-45.762,179.672,4.020,148.741
C06677=1120.591,-121.451,-45.753,179.672,4.015,148.740
C06678=1120.596,-121.700,-45.746,179.673,4.009,148.738
C06679=1120.602,-121.950,-45.737,179.673,4.004,148.737
C06680=1120.608,-122.200,-45.729,179.673,3.998,148.736
C06681=1120.613,-122.451,-45.721,179.673,3.993,148.735
C06682=1120.618,-122.699,-45.713,179.673,3.988,148.733
C06683=1120.624,-122.950,-45.705,179.674,3.983,148.732
C06684=1120.629,-123.200,-45.696,179.674,3.976,148.731
C06685=1120.634,-123.449,-45.689,179.674,3.971,148.729
C06686=1120.640,-123.700,-45.681,179.675,3.966,148.728
C06687=1120.645,-123.949,-45.672,179.675,3.961,148.727
C06688=1120.651,-124.199,-45.664,179.675,3.955,148.726
C06689=1120.656,-124.448,-45.656,179.675,3.950,148.725
C06690=1120.661,-124.699,-45.648,179.676,3.944,148.723
C06691=1120.667,-124.948,-45.640,179.676,3.939,148.722
C06692=1120.672,-125.198,-45.632,179.676,3.933,148.721
C06693=1120.678,-125.448,-45.624,179.676,3.928,148.720
C06694=1120.683,-125.698,-45.616,179.676,3.923,148.718
C06695=1120.688,-125.947,-45.608,179.677,3.916,148.717
C06696=1120.694,-126.197,-45.600,179.677,3.911,148.716
C06697=1120.700,-126.447,-45.592,179.677,3.906,148.714
C06698=1120.704,-126.697,-45.584,179.677,3.900,148.713
C06699=1120.710,-126.946,-45.576,179.678,3.894,148.712
C06700=1120.715,-127.197,-45.568,179.678,3.889,148.711
C06701=1120.721,-127.446,-45.560,179.678,3.883,148.709
C06702=1120.726,-127.696,-45.552,179.678,3.878,148.708
C06703=1120.732,-127.946,-45.544,179.679,3.872,148.707
C06704=1120.738,-128.195,-45.537,179.679,3.866,148.705
C06705=1120.743,-128.446,-45.529,179.679,3.861,148.704
C06706=1120.749,-128.695,-45.521,179.680,3.856,148.703
C06707=1120.325,-128.686,-45.546,179.686,3.859,148.702
C06708=1120.321,-128.470,-45.554,179.686,3.865,148.703
C06709=1120.316,-128.254,-45.560,179.686,3.869,148.704
C06710=1120.311,-128.039,-45.568,179.686,3.875,148.705
C06711=1120.306,-127.824,-45.574,179.686,3.879,148.706
C06712=1120.302,-127.608,-45.581,179.685,3.884,148.707
C06713=1120.297,-127.392,-45.588,179.686,3.889,148.708
C06714=1120.292,-127.177,-45.594,179.685,3.894,148.709
C06715=1120.288,-126.962,-45.602,179.685,3.898,148.710
C06716=1120.282,-126.712,-45.610,179.685,3.904,148.712
C06717=1120.277,-126.462,-45.617,179.684,3.909,148.713
C06718=1120.272,-126.212,-45.626,179.684,3.914,148.714
C06719=1120.266,-125.962,-45.634,179.684,3.920,148.715
C06720=1120.261,-125.712,-45.641,179.683,3.926,148.717
C06721=1120.255,-125.463,-45.650,179.683,3.931,148.718
C06722=1120.250,-125.213,-45.658,179.683,3.936,148.719
C06723=1120.244,-124.963,-45.665,179.683,3.942,148.720
C06724=1120.239,-124.713,-45.674,179.682,3.948,148.722
C06725=1120.234,-124.463,-45.682,179.682,3.953,148.723
C06726=1120.229,-124.214,-45.690,179.682,3.959,148.724
C06727=1120.223,-123.964,-45.698,179.682,3.964,148.726
C06728=1120.217,-123.714,-45.706,179.682,3.969,148.727
C06729=1120.212,-123.464,-45.715,179.681,3.975,148.728
C06730=1120.206,-123.214,-45.722,179.681,3.981,148.729
C06731=1120.201,-122.965,-45.731,179.681,3.986,148.731
C06732=1120.195,-122.715,-45.739,179.681,3.991,148.732
C06733=1120.191,-122.465,-45.747,179.680,3.996,148.733
C06734=1120.185,-122.216,-45.755,179.680,4.002,148.734
C06735=1120.179,-121.965,-45.763,179.680,4.008,148.736
C06736=1120.174,-121.715,-45.772,179.680,4.013,148.737
C06737=1120.168,-121.465,-45.780,179.679,4.018,148.738
C06738=1120.164,-121.216,-45.788,179.679,4.024,148.739
C06739=1120.158,-120.966,-45.796,179.679,4.029,148.741
C06740=1120.152,-120.716,-45.805,179.679,4.035,148.742
C06741=1120.147,-120.466,-45.813,179.679,4.040,148.743
C06742=1120.142,-120.217,-45.821,179.678,4.045,148.744
C06743=1120.137,-119.967,-45.830,179.678,4.051,148.746
C06744=1120.131,-119.717,-45.838,179.677,4.056,148.747
C06745=1120.125,-119.468,-45.847,179.678,4.062,148.748
C06746=1120.120,-119.217,-45.855,179.677,4.067,148.749
C06747=1120.114,-118.968,-45.864,179.677,4.072,148.750
C06748=1120.109,-118.718,-45.871,179.677,4.077,148.752
C06749=1120.104,-118.468,-45.880,179.676,4.082,148.753
C06750=1120.099,-118.219,-45.889,179.676,4.088,148.754
C06751=1120.093,-117.968,-45.897,179.676,4.093,148.755
C06752=1120.088,-117.718,-45.906,179.675,4.098,148.757
C06753=1120.082,-117.469,-45.913,179.675,4.104,148.758
C06754=1120.077,-117.219,-45.922,179.675,4.110,148.759
C06755=1120.072,-116.970,-45.930,179.675,4.115,148.760
C06756=1120.066,-116.719,-45.938,179.675,4.120,148.762
C06757=1120.061,-116.470,-45.947,179.674,4.125,148.763
C06758=1120.055,-116.221,-45.956,179.674,4.130,148.764
C06759=1120.050,-115.970,-45.964,179.674,4.135,148.765
C06760=1120.045,-115.720,-45.973,179.674,4.141,148.766
C06761=1120.039,-115.471,-45.982,179.673,4.146,148.768
C06762=1120.033,-115.221,-45.990,179.673,4.151,148.769
C06763=1120.028,-114.971,-45.999,179.673,4.157,148.770
C06764=1120.023,-114.756,-46.006,179.672,4.161,148.771
C06765=1120.018,-114.540,-46.013,179.673,4.166,148.772
C06766=1120.015,-114.324,-46.020,179.672,4.170,148.773
C06767=1120.010,-114.109,-46.028,179.672,4.175,148.774
C06768=1120.005,-113.894,-46.035,179.672,4.179,148.775
C06769=1120.000,-113.678,-46.043,179.671,4.183,148.776
C06770=1119.996,-113.463,-46.051,179.671,4.188,148.777
C06771=1119.991,-113.247,-46.057,179.671,4.192,148.778
C06772=1119.986,-112.997,-46.066,179.671,4.197,148.780
C06773=1119.980,-112.747,-46.075,179.671,4.203,148.781
C06774=1119.975,-112.498,-46.084,179.671,4.209,148.782
C06775=1119.969,-112.248,-46.093,179.670,4.214,148.783
C06776=1119.964,-111.998,-46.101,179.670,4.219,148.784
C06777=1119.958,-111.749,-46.109,179.670,4.224,148.786
C06778=1119.953,-111.499,-46.118,179.670,4.229,148.787
C06779=1119.948,-111.249,-46.127,179.669,4.234,148.788
C06780=1119.943,-110.999,-46.136,179.669,4.240,148.789
C06781=1119.937,-110.750,-46.145,179.669,4.245,148.790
C06782=1119.931,-110.499,-46.153,179.669,4.250,148.792
C06783=1119.926,-110.250,-46.162,179.668,4.254,148.793
C06784=1119.921,-110.000,-46.171,179.668,4.259,148.794
C06785=1119.916,-109.750,-46.180,179.667,4.265,148.795
C06786=1119.910,-109.501,-46.188,179.667,4.270,148.796
C06787=1119.905,-109.251,-46.197,179.667,4.275,148.798
C06788=1119.900,-109.001,-46.206,179.667,4.280,148.799
C06789=1119.895,-108.751,-46.215,179.666,4.285,148.800
C06790=1119.889,-108.501,-46.223,179.666,4.290,148.801
C06791=1119.883,-108.252,-46.231,179.666,4.296,148.802
C06792=1119.878,-108.002,-46.240,179.666,4.301,148.804
C06793=1119.872,-107.752,-46.250,179.665,4.306,148.805
C06794=1119.867,-107.502,-46.259,179.665,4.311,148.806
C06795=1119.862,-107.252,-46.268,179.665,4.316,148.807
C06796=1119.856,-107.003,-46.276,179.665,4.321,148.808
C06797=1119.851,-106.753,-46.285,179.664,4.327,148.810
C06798=1119.846,-106.503,-46.294,179.664,4.332,148.811
C06799=1119.841,-106.253,-46.303,179.664,4.337,148.812
C06800=1119.836,-106.003,-46.312,179.664,4.341,148.813
C06801=1119.830,-105.753,-46.321,179.663,4.346,148.814
C06802=1119.824,-105.504,-46.330,179.663,4.351,148.815
C06803=1119.819,-105.254,-46.339,179.663,4.356,148.817
C06804=1119.814,-105.004,-46.348,179.663,4.362,148.818
C06805=1119.808,-104.754,-46.357,179.662,4.367,148.819
C06806=1119.803,-104.505,-46.365,179.662,4.372,148.820
C06807=1119.797,-104.254,-46.375,179.662,4.377,148.821
C06808=1119.792,-104.005,-46.384,179.662,4.382,148.823
C06809=1119.787,-103.755,-46.393,179.661,4.387,148.824
C06810=1119.782,-103.506,-46.402,179.661,4.392,148.825
C06811=1119.776,-103.256,-46.411,179.660,4.397,148.826
C06812=1119.771,-103.007,-46.420,179.660,4.402,148.827
C06813=1119.765,-102.756,-46.429,179.660,4.407,148.829
C06814=1119.760,-102.507,-46.438,179.660,4.412,148.830
C06815=1119.755,-102.257,-46.447,179.660,4.418,148.831
C06816=1119.750,-102.007,-46.456,179.659,4.422,148.832
C06817=1119.744,-101.757,-46.465,179.658,4.427,148.833
C06818=1119.739,-101.507,-46.474,179.659,4.432,148.834
C06819=1119.734,-101.258,-46.484,179.659,4.437,148.835
C06820=1119.729,-101.042,-46.492,179.658,4.441,148.837
C06821=1119.724,-100.827,-46.499,179.657,4.445,148.838
C06822=1119.720,-100.612,-46.507,179.658,4.450,148.839
C06823=1119.715,-100.396,-46.515,179.657,4.454,148.839
C06824=1119.710,-100.180,-46.523,179.657,4.459,148.841
C06825=1119.705,-99.965,-46.531,179.657,4.463,148.842
C06826=1119.701,-99.749,-46.539,179.657,4.467,148.843
C06827=1119.696,-99.534,-46.547,179.656,4.471,148.844
C06828=1119.692,-99.285,-46.556,179.656,4.476,148.845
C06829=1119.686,-99.035,-46.566,179.656,4.482,148.846
C06830=1119.681,-98.785,-46.575,179.656,4.487,148.847
C06831=1119.675,-98.535,-46.583,179.655,4.491,148.848
C06832=1119.670,-98.285,-46.592,179.655,4.496,148.849
C06833=1119.665,-98.036,-46.603,179.654,4.501,148.851
C06834=1119.659,-97.786,-46.611,179.654,4.507,148.852
C06835=1119.654,-97.536,-46.620,179.653,4.511,148.853
C06836=1119.648,-97.286,-46.630,179.653,4.516,148.854
C06837=1119.644,-97.037,-46.639,179.653,4.521,148.855
C06838=1119.638,-96.788,-46.648,179.653,4.526,148.857
C06839=1119.632,-96.537,-46.657,179.653,4.532,148.858
C06840=1119.627,-96.288,-46.667,179.652,4.536,148.859
C06841=1119.621,-96.038,-46.677,179.652,4.541,148.860
C06842=1119.616,-95.788,-46.685,179.652,4.546,148.861
C06843=1119.611,-95.539,-46.695,179.652,4.551,148.862
C06844=1119.605,-95.289,-46.705,179.651,4.555,148.863
C06845=1119.600,-95.039,-46.713,179.651,4.561,148.865
C06846=1119.595,-94.790,-46.723,179.650,4.566,148.866
C06847=1119.589,-94.540,-46.733,179.650,4.571,148.867
C06848=1119.584,-94.290,-46.741,179.649,4.575,148.868
C06849=1119.579,-94.039,-46.752,179.649,4.580,148.869
C06850=1119.574,-93.790,-46.761,179.648,4.585,148.871
C06851=1119.568,-93.539,-46.770,179.647,4.589,148.872
C06852=1119.563,-93.290,-46.780,179.647,4.595,148.873
C06853=1119.558,-93.040,-46.789,179.646,4.599,148.874
C06854=1119.552,-92.791,-46.799,179.646,4.604,148.876
C06855=1119.547,-92.541,-46.808,179.645,4.609,148.877
C06856=1119.541,-92.291,-46.818,179.644,4.613,148.878
C06857=1119.536,-92.042,-46.827,179.644,4.618,148.879
C06858=1119.531,-91.791,-46.837,179.643,4.623,148.881
C06859=1119.526,-91.542,-46.846,179.643,4.628,148.882
C06860=1119.520,-91.292,-46.855,179.641,4.633,148.883
C06861=1119.515,-91.043,-46.865,179.641,4.638,148.884
C06862=1119.510,-90.793,-46.874,179.640,4.642,148.886
C06863=1119.504,-90.543,-46.884,179.640,4.647,148.887
C06864=1119.499,-90.294,-46.893,179.640,4.652,148.888
C06865=1119.493,-90.043,-46.903,179.639,4.657,148.889
C06866=1119.488,-89.794,-46.912,179.639,4.662,148.891
C06867=1119.482,-89.544,-46.922,179.638,4.667,148.892
C06868=1119.478,-89.294,-46.932,179.638,4.672,148.893
C06869=1119.472,-89.044,-46.941,179.637,4.677,148.894
C06870=1119.467,-88.795,-46.951,179.637,4.681,148.895
C06871=1119.461,-88.545,-46.961,179.636,4.687,148.897
C06872=1119.456,-88.295,-46.970,179.635,4.691,148.898
C06873=1119.451,-88.045,-46.980,179.635,4.696,148.899
C06874=1119.446,-87.796,-46.989,179.635,4.702,148.900
C06875=1119.440,-87.546,-46.999,179.634,4.706,148.901
C06876=1119.436,-87.331,-47.007,179.634,4.711,148.903
C06877=1119.431,-87.115,-47.015,179.634,4.715,148.904
C06878=1119.426,-86.900,-47.024,179.633,4.719,148.905
C06879=1119.422,-86.685,-47.032,179.633,4.723,148.906
C06880=1119.418,-86.470,-47.041,179.632,4.728,148.907
C06881=1119.413,-86.254,-47.049,179.632,4.733,148.908
C06882=1119.408,-86.039,-47.058,179.631,4.737,148.909
C06883=1119.404,-85.823,-47.066,179.631,4.741,148.910
C06884=1119.398,-85.574,-47.076,179.631,4.746,148.911
C06885=1119.393,-85.324,-47.085,179.631,4.751,148.912
C06886=1119.388,-85.074,-47.095,179.630,4.755,148.913
C06887=1119.382,-84.825,-47.105,179.629,4.761,148.915
C06888=1119.377,-84.575,-47.114,179.629,4.766,148.916
C06889=1119.372,-84.325,-47.125,179.629,4.771,148.917
C06890=1119.367,-84.075,-47.134,179.629,4.776,148.918
C06891=1119.361,-83.825,-47.144,179.629,4.782,148.920
C06892=1119.356,-83.576,-47.154,179.628,4.786,148.921
C06893=1119.351,-83.327,-47.163,179.628,4.791,148.922
C06894=1119.345,-83.076,-47.173,179.627,4.796,148.923
C06895=1119.340,-82.826,-47.184,179.627,4.801,148.924
C06896=1119.335,-82.577,-47.193,179.627,4.807,148.926
C06897=1119.329,-82.327,-47.203,179.626,4.812,148.927
C06898=1119.324,-82.078,-47.212,179.626,4.817,148.928
C06899=1119.319,-81.828,-47.222,179.626,4.822,148.929
C06900=1119.313,-81.578,-47.232,179.625,4.827,148.930
C06901=1119.308,-81.328,-47.242,179.625,4.832,148.932
C06902=1119.303,-81.078,-47.252,179.625,4.837,148.933
C06903=1119.297,-80.829,-47.262,179.625,4.842,148.934
C06904=1119.292,-80.579,-47.271,179.625,4.847,148.935
C06905=1119.287,-80.329,-47.282,179.625,4.853,148.936
C06906=1119.281,-80.079,-47.292,179.624,4.858,148.937
C06907=1119.276,-79.830,-47.302,179.624,4.863,148.939
C06908=1119.271,-79.580,-47.311,179.624,4.868,148.940
C06909=1119.265,-79.330,-47.321,179.624,4.873,148.941
C06910=1119.260,-79.080,-47.332,179.624,4.878,148.942
C06911=1119.255,-78.831,-47.342,179.624,4.884,148.943
C06912=1119.250,-78.581,-47.352,179.623,4.889,148.944
C06913=1119.244,-78.332,-47.362,179.623,4.894,148.946
C06914=1119.239,-78.081,-47.372,179.623,4.899,148.947
C06915=1119.233,-77.831,-47.382,179.623,4.904,148.948
C06916=1119.228,-77.582,-47.392,179.623,4.909,148.949
C06917=1119.223,-77.332,-47.402,179.623,4.915,148.950
C06918=1119.218,-77.082,-47.412,179.623,4.920,148.951
C06919=1119.212,-76.833,-47.423,179.623,4.926,148.953
C06920=1119.207,-76.583,-47.432,179.623,4.931,148.954
C06921=1119.201,-76.333,-47.442,179.623,4.936,148.955
C06922=1119.196,-76.083,-47.452,179.623,4.941,148.956
C06923=1119.191,-75.834,-47.463,179.623,4.946,148.957
C06924=1119.185,-75.584,-47.473,179.623,4.951,148.958
C06925=1119.181,-75.334,-47.483,179.623,4.956,148.959
C06926=1119.175,-75.084,-47.493,179.623,4.962,148.960
C06927=1119.170,-74.835,-47.503,179.623,4.967,148.962
C06928=1119.164,-74.585,-47.513,179.623,4.972,148.963
C06929=1119.159,-74.335,-47.524,179.623,4.977,148.964
C06930=1119.153,-74.086,-47.534,179.623,4.982,148.965
C06931=1119.148,-73.836,-47.544,179.623,4.987,148.966
C06932=1119.144,-73.621,-47.553,179.623,4.992,148.967
C06933=1119.139,-73.405,-47.562,179.623,4.997,148.968
C06934=1119.135,-73.190,-47.570,179.623,5.001,148.969
C06935=1119.130,-72.975,-47.579,179.624,5.006,148.970
C06936=1119.126,-72.760,-47.588,179.623,5.011,148.971
C06937=1119.121,-72.545,-47.597,179.623,5.015,148.972
C06938=1119.116,-72.329,-47.606,179.624,5.020,148.973
C06939=1119.112,-72.114,-47.615,179.624,5.024,148.974
C06940=1119.107,-71.865,-47.625,179.624,5.029,148.975
C06941=1119.102,-71.614,-47.636,179.624,5.034,148.976
C06942=1119.096,-71.365,-47.646,179.624,5.039,148.977
C06943=1119.090,-71.115,-47.656,179.624,5.045,148.978
C06944=1119.085,-70.865,-47.667,179.625,5.050,148.979
C06945=1119.080,-70.616,-47.678,179.625,5.055,148.980
C06946=1119.074,-70.367,-47.688,179.625,5.060,148.981
C06947=1119.069,-70.116,-47.698,179.626,5.066,148.982
C06948=1119.064,-69.867,-47.709,179.625,5.071,148.983
C06949=1119.059,-69.617,-47.719,179.626,5.076,148.984
C06950=1119.053,-69.367,-47.729,179.626,5.082,148.986
C06951=1119.048,-69.117,-47.740,179.627,5.087,148.986
C06952=1119.043,-68.868,-47.751,179.626,5.092,148.988
C06953=1119.037,-68.618,-47.761,179.627,5.098,148.989
C06954=1119.032,-68.368,-47.772,179.627,5.102,148.990
C06955=1119.027,-68.119,-47.782,179.627,5.108,148.991
C06956=1119.022,-67.868,-47.792,179.628,5.113,148.992
C06957=1119.017,-67.619,-47.803,179.628,5.118,148.993
C06958=1119.012,-67.369,-47.814,179.628,5.123,148.994
C06959=1119.006,-67.120,-47.824,179.629,5.129,148.995
C06960=1119.000,-66.870,-47.834,179.629,5.134,148.996
C06961=1118.996,-66.620,-47.846,179.630,5.139,148.997
C06962=1118.990,-66.371,-47.856,179.630,5.145,148.998
C06963=1118.985,-66.121,-47.866,179.630,5.149,148.999
C06964=1118.979,-65.871,-47.877,179.631,5.155,149.000
C06965=1118.975,-65.621,-47.888,179.631,5.160,149.001
C06966=1118.969,-65.372,-47.898,179.632,5.166,149.002
C06967=1118.964,-65.122,-47.909,179.632,5.171,149.003
C06968=1118.959,-64.873,-47.920,179.633,5.175,149.004
C06969=1118.954,-64.622,-47.930,179.634,5.181,149.005
C06970=1118.948,-64.373,-47.941,179.634,5.186,149.006
C06971=1118.943,-64.123,-47.952,179.634,5.192,149.007
C06972=1118.937,-63.873,-47.962,179.635,5.196,149.008
C06973=1118.933,-63.624,-47.974,179.636,5.202,149.009
C06974=1118.927,-63.374,-47.984,179.636,5.207,149.010
C06975=1118.922,-63.124,-47.995,179.636,5.212,149.011
C06976=1118.917,-62.874,-48.006,179.637,5.218,149.012
C06977=1118.912,-62.625,-48.016,179.637,5.222,149.013
C06978=1118.906,-62.375,-48.028,179.638,5.228,149.014
C06979=1118.901,-62.125,-48.038,179.639,5.233,149.015
C06980=1118.896,-61.876,-48.049,179.640,5.238,149.016
C06981=1118.890,-61.626,-48.060,179.640,5.243,149.016
C06982=1118.886,-61.377,-48.071,179.641,5.249,149.018
C06983=1118.880,-61.126,-48.082,179.641,5.254,149.019
C06984=1118.875,-60.877,-48.093,179.642,5.259,149.019
C06985=1118.870,-60.627,-48.104,179.642,5.264,149.020
C06986=1118.864,-60.378,-48.114,179.643,5.270,149.021
C06987=1118.859,-60.128,-48.125,179.644,5.274,149.022
C06988=1118.855,-59.913,-48.135,179.644,5.278,149.023
C06989=1118.850,-59.697,-48.144,179.644,5.283,149.024
C06990=1118.846,-59.482,-48.154,179.644,5.287,149.025
C06991=1118.841,-59.268,-48.163,179.644,5.290,149.026
C06992=1118.836,-59.052,-48.173,179.644,5.294,149.027
C06993=1118.832,-58.837,-48.183,179.644,5.298,149.027
C06994=1118.827,-58.622,-48.192,179.643,5.302,149.028
C06995=1118.822,-58.406,-48.201,179.643,5.306,149.029
C06996=1118.818,-58.157,-48.212,179.643,5.311,149.030
C06997=1118.813,-57.908,-48.223,179.642,5.316,149.032
C06998=1118.808,-57.658,-48.234,179.643,5.321,149.033
C06999=1118.802,-57.408,-48.246,179.642,5.325,149.034
C07000=1118.796,-57.158,-48.256,179.642,5.330,149.035
C07001=1118.792,-56.908,-48.267,179.642,5.335,149.036
C07002=1118.786,-56.659,-48.279,179.642,5.339,149.037
C07003=1118.781,-56.409,-48.289,179.642,5.344,149.038
C07004=1118.776,-56.159,-48.301,179.641,5.348,149.039
C07005=1118.770,-55.910,-48.312,179.641,5.353,149.040
C07006=1118.765,-55.660,-48.323,179.642,5.358,149.041
C07007=1118.760,-55.410,-48.334,179.641,5.362,149.042
C07008=1118.756,-55.161,-48.345,179.641,5.368,149.043
C07009=1118.750,-54.911,-48.357,179.641,5.372,149.044
C07010=1118.745,-54.661,-48.367,179.641,5.377,149.045
C07011=1118.739,-54.411,-48.379,179.641,5.382,149.047
C07012=1118.734,-54.162,-48.390,179.640,5.386,149.048
C07013=1118.729,-53.912,-48.401,179.640,5.391,149.049
C07014=1118.723,-53.662,-48.413,179.640,5.395,149.050
C07015=1118.718,-53.413,-48.424,179.640,5.400,149.051
C07016=1118.713,-53.164,-48.435,179.639,5.404,149.052
C07017=1118.708,-52.913,-48.446,179.639,5.409,149.053
C07018=1118.702,-52.664,-48.457,179.640,5.414,149.054
C07019=1118.697,-52.414,-48.469,179.639,5.419,149.055
C07020=1118.692,-52.165,-48.480,179.639,5.424,149.056
C07021=1118.687,-51.914,-48.491,179.639,5.428,149.057
C07022=1118.681,-51.665,-48.502,179.639,5.433,149.058
C07023=1118.677,-51.415,-48.514,179.639,5.438,149.059
C07024=1118.671,-51.165,-48.526,179.638,5.442,149.061
C07025=1118.666,-50.916,-48.537,179.638,5.447,149.062
C07026=1118.660,-50.667,-48.548,179.638,5.451,149.063
C07027=1118.655,-50.416,-48.559,179.638,5.456,149.064
C07028=1118.650,-50.166,-48.571,179.638,5.461,149.065
C07029=1118.645,-49.918,-48.582,179.637,5.466,149.066
C07030=1118.640,-49.668,-48.593,179.637,5.471,149.067
C07031=1118.635,-49.418,-48.605,179.637,5.475,149.068
C07032=1118.630,-49.168,-48.616,179.637,5.480,149.069
C07033=1118.624,-48.918,-48.627,179.637,5.485,149.070
C07034=1118.619,-48.669,-48.638,179.636,5.489,149.071
C07035=1118.613,-48.419,-48.650,179.637,5.494,149.072
C07036=1118.609,-48.169,-48.661,179.636,5.498,149.073
C07037=1118.603,-47.919,-48.673,179.636,5.503,149.075
C07038=1118.598,-47.670,-48.684,179.636,5.508,149.076
C07039=1118.593,-47.420,-48.696,179.636,5.513,149.077
C07040=1118.588,-47.171,-48.707,179.636,5.518,149.078
C07041=1118.583,-46.921,-48.719,179.635,5.522,149.079
C07042=1118.576,-46.672,-48.731,179.635,5.527,149.080
C07043=1118.572,-46.422,-48.742,179.635,5.532,149.081
C07044=1118.567,-46.207,-48.751,179.635,5.536,149.082
C07045=1118.563,-45.992,-48.761,179.635,5.540,149.083
C07046=1118.558,-45.777,-48.771,179.635,5.544,149.084
C07047=1118.553,-45.562,-48.782,179.635,5.548,149.085
C07048=1118.549,-45.347,-48.792,179.634,5.552,149.086
C07049=1118.544,-45.131,-48.801,179.634,5.556,149.086
C07050=1118.540,-44.916,-48.811,179.634,5.560,149.088
C07051=1118.536,-44.702,-48.821,179.633,5.564,149.089
C07052=1118.530,-44.452,-48.833,179.634,5.569,149.089
C07053=1118.526,-44.202,-48.845,179.634,5.574,149.091
C07054=1118.520,-43.952,-48.856,179.633,5.578,149.092
C07055=1118.515,-43.702,-48.868,179.633,5.583,149.093
C07056=1118.509,-43.453,-48.879,179.633,5.587,149.094
C07057=1118.504,-43.203,-48.891,179.633,5.592,149.095
C07058=1118.499,-42.954,-48.902,179.633,5.597,149.096
C07059=1118.494,-42.704,-48.914,179.634,5.603,149.097
C07060=1118.488,-42.454,-48.926,179.635,5.608,149.098
C07061=1118.484,-42.204,-48.937,179.637,5.613,149.098
C07062=1118.479,-41.955,-48.950,179.638,5.619,149.099
C07063=1118.474,-41.705,-48.961,179.639,5.624,149.100
C07064=1118.468,-41.456,-48.973,179.641,5.630,149.101
C07065=1118.463,-41.206,-48.985,179.642,5.635,149.102
C07066=1118.458,-40.956,-48.996,179.643,5.640,149.102
C07067=1118.452,-40.706,-49.008,179.644,5.646,149.103
C07068=1118.447,-40.457,-49.020,179.645,5.651,149.104
C07069=1118.442,-40.207,-49.032,179.647,5.657,149.105
C07070=1118.437,-39.958,-49.044,179.647,5.661,149.106
C07071=1118.432,-39.708,-49.056,179.649,5.666,149.106
C07072=1118.426,-39.458,-49.067,179.650,5.672,149.107
C07073=1118.421,-39.208,-49.080,179.650,5.677,149.108
C07074=1118.416,-38.959,-49.091,179.652,5.682,149.109
C07075=1118.410,-38.710,-49.103,179.652,5.687,149.110
C07076=1118.405,-38.460,-49.115,179.654,5.692,149.110
C07077=1118.400,-38.210,-49.127,179.654,5.697,149.111
C07078=1118.395,-37.961,-49.139,179.655,5.701,149.112
C07079=1118.390,-37.711,-49.151,179.656,5.706,149.113
C07080=1118.385,-37.461,-49.163,179.657,5.711,149.114
C07081=1118.379,-37.211,-49.175,179.657,5.716,149.115
C07082=1118.374,-36.962,-49.187,179.659,5.721,149.115
C07083=1118.369,-36.713,-49.199,179.659,5.726,149.116
C07084=1118.364,-36.463,-49.211,179.660,5.730,149.117
C07085=1118.359,-36.213,-49.223,179.660,5.735,149.118
C07086=1118.353,-35.963,-49.235,179.661,5.740,149.119
C07087=1118.348,-35.713,-49.247,179.662,5.744,149.119
C07088=1118.343,-35.463,-49.259,179.662,5.749,149.120
C07089=1118.338,-35.214,-49.271,179.663,5.753,149.121
C07090=1118.333,-34.965,-49.283,179.664,5.758,149.122
C07091=1118.328,-34.715,-49.296,179.664,5.763,149.123
C07092=1118.322,-34.465,-49.307,179.664,5.767,149.124
C07093=1118.317,-34.216,-49.320,179.665,5.772,149.125
C07094=1118.312,-33.966,-49.332,179.665,5.777,149.126
C07095=1118.307,-33.717,-49.344,179.666,5.780,149.126
C07096=1118.302,-33.466,-49.357,179.666,5.785,149.127
C07097=1118.296,-33.216,-49.369,179.667,5.790,149.128
C07098=1118.291,-32.967,-49.381,179.667,5.794,149.129
C07099=1118.286,-32.717,-49.393,179.667,5.799,149.130
C07100=1118.282,-32.503,-49.404,179.667,5.802,149.131
C07101=1118.277,-32.288,-49.414,179.667,5.806,149.131
C07102=1118.272,-32.073,-49.424,179.668,5.810,149.132
C07103=1118.268,-31.858,-49.435,179.667,5.814,149.133
C07104=1118.264,-31.642,-49.446,179.668,5.817,149.134
C07105=1118.259,-31.428,-49.456,179.668,5.821,149.135
C07106=1118.255,-31.213,-49.467,179.668,5.825,149.135
C07107=1118.250,-30.998,-49.477,179.668,5.828,149.136
C07108=1118.245,-30.748,-49.489,179.668,5.833,149.137
C07109=1118.240,-30.499,-49.502,179.668,5.837,149.138
C07110=1118.235,-30.249,-49.515,179.668,5.841,149.139
C07111=1118.230,-29.999,-49.527,179.668,5.846,149.140
C07112=1118.225,-29.750,-49.539,179.668,5.850,149.141
C07113=1118.219,-29.500,-49.551,179.668,5.854,149.142
C07114=1118.214,-29.250,-49.564,179.668,5.859,149.143
C07115=1118.209,-29.001,-49.576,179.668,5.863,149.144
C07116=1118.204,-28.751,-49.588,179.667,5.867,149.145
C07117=1118.198,-28.502,-49.601,179.667,5.871,149.146
C07118=1118.193,-28.252,-49.613,179.667,5.875,149.147
C07119=1118.188,-28.002,-49.626,179.666,5.879,149.148
C07120=1118.183,-27.753,-49.638,179.666,5.884,149.149
C07121=1118.178,-27.503,-49.650,179.666,5.888,149.150
C07122=1118.173,-27.253,-49.663,179.665,5.892,149.151
C07123=1118.168,-27.004,-49.676,179.664,5.896,149.152
C07124=1118.162,-26.754,-49.687,179.664,5.900,149.153
C07125=1118.157,-26.505,-49.700,179.664,5.905,149.154
C07126=1118.153,-26.255,-49.713,179.663,5.909,149.155
C07127=1118.147,-26.005,-49.725,179.662,5.913,149.156
C07128=1118.142,-25.755,-49.737,179.662,5.917,149.157
C07129=1118.137,-25.506,-49.750,179.663,5.923,149.158
C07130=1118.132,-25.257,-49.763,179.664,5.927,149.159
C07131=1118.126,-25.007,-49.775,179.664,5.932,149.160
C07132=1118.122,-24.757,-49.788,179.665,5.937,149.161
C07133=1118.117,-24.508,-49.800,179.665,5.942,149.162
C07134=1118.111,-24.257,-49.813,179.666,5.946,149.163
C07135=1118.105,-24.008,-49.825,179.667,5.952,149.164
C07136=1118.100,-23.759,-49.838,179.667,5.957,149.164
C07137=1118.096,-23.509,-49.851,179.668,5.961,149.165
C07138=1118.090,-23.259,-49.863,179.668,5.966,149.166
C07139=1118.085,-23.009,-49.875,179.669,5.971,149.167
C07140=1118.080,-22.760,-49.888,179.669,5.976,149.168
C07141=1118.074,-22.510,-49.901,179.670,5.980,149.169
C07142=1118.070,-22.260,-49.914,179.670,5.985,149.170
C07143=1118.065,-22.011,-49.927,179.672,5.990,149.170
C07144=1118.059,-21.761,-49.938,179.672,5.995,149.171
C07145=1118.054,-21.512,-49.951,179.673,6.000,149.172
C07146=1118.049,-21.263,-49.964,179.673,6.004,149.173
C07147=1118.044,-21.012,-49.977,179.674,6.009,149.174
C07148=1118.039,-20.763,-49.990,179.674,6.014,149.175
C07149=1118.033,-20.514,-50.002,179.675,6.019,149.176
C07150=1118.028,-20.264,-50.015,179.675,6.023,149.177
C07151=1118.024,-20.014,-50.028,179.676,6.028,149.177
C07152=1118.018,-19.765,-50.041,179.677,6.032,149.178
C07153=1118.012,-19.515,-50.053,179.677,6.037,149.179
C07154=1118.007,-19.265,-50.066,179.678,6.043,149.180
C07155=1118.003,-19.015,-50.079,179.679,6.047,149.181
C07156=1117.998,-18.801,-50.090,179.679,6.051,149.182
C07157=1117.993,-18.586,-50.101,179.680,6.055,149.182
C07158=1117.990,-18.371,-50.112,179.680,6.059,149.183
C07159=1117.985,-18.156,-50.123,179.681,6.063,149.184
C07160=1117.980,-17.942,-50.134,179.681,6.067,149.185
C07161=1117.976,-17.726,-50.146,179.682,6.071,149.185
C07162=1117.971,-17.511,-50.156,179.682,6.075,149.186
C07163=1117.967,-17.297,-50.167,179.682,6.079,149.187
C07164=1117.962,-17.047,-50.180,179.683,6.084,149.188
C07165=1117.956,-16.797,-50.193,179.685,6.089,149.188
C07166=1117.951,-16.548,-50.206,179.685,6.093,149.189
C07167=1117.947,-16.298,-50.219,179.686,6.098,149.190
C07168=1117.941,-16.048,-50.232,179.686,6.103,149.191
C07169=1117.936,-15.800,-50.246,179.686,6.108,149.192
C07170=1117.931,-15.549,-50.259,179.687,6.112,149.193
C07171=1117.926,-15.300,-50.272,179.688,6.117,149.193
C07172=1117.921,-15.051,-50.284,179.688,6.121,149.194
C07173=1117.916,-14.801,-50.297,179.689,6.126,149.195
C07174=1117.910,-14.551,-50.310,179.690,6.131,149.196
C07175=1117.906,-14.301,-50.323,179.690,6.135,149.197
C07176=1117.900,-14.052,-50.336,179.691,6.140,149.198
C07177=1117.895,-13.803,-50.350,179.691,6.145,149.199
C07178=1117.890,-13.553,-50.363,179.692,6.149,149.199
C07179=1117.885,-13.303,-50.376,179.693,6.154,149.200
C07180=1117.879,-13.054,-50.389,179.693,6.158,149.201
C07181=1117.875,-12.804,-50.402,179.694,6.162,149.202
C07182=1117.869,-12.554,-50.415,179.694,6.167,149.203
C07183=1117.865,-12.305,-50.429,179.695,6.172,149.204
C07184=1117.859,-12.055,-50.442,179.695,6.176,149.204
C07185=1117.854,-11.805,-50.455,179.696,6.181,149.205
C07186=1117.849,-11.555,-50.468,179.697,6.185,149.206
C07187=1117.844,-11.307,-50.481,179.697,6.190,149.207
C07188=1117.839,-11.057,-50.494,179.698,6.195,149.208
C07189=1117.833,-10.807,-50.507,179.699,6.199,149.208
C07190=1117.829,-10.557,-50.520,179.699,6.204,149.209
C07191=1117.823,-10.308,-50.534,179.700,6.209,149.210
C07192=1117.819,-10.058,-50.547,179.701,6.213,149.211
C07193=1117.813,-9.808,-50.560,179.701,6.218,149.212
C07194=1117.809,-9.559,-50.574,179.702,6.222,149.213
C07195=1117.803,-9.309,-50.587,179.703,6.227,149.213
C07196=1117.798,-9.060,-50.600,179.703,6.231,149.214
C07197=1117.793,-8.810,-50.614,179.704,6.236,149.215
C07198=1117.788,-8.561,-50.627,179.704,6.241,149.216
C07199=1117.782,-8.311,-50.640,179.705,6.245,149.217
C07200=1117.778,-8.062,-50.654,179.705,6.249,149.218
C07201=1117.772,-7.812,-50.667,179.706,6.254,149.218
C07202=1117.767,-7.563,-50.681,179.707,6.258,149.219
C07203=1117.762,-7.312,-50.694,179.707,6.263,149.220
C07204=1117.756,-7.063,-50.707,179.708,6.268,149.221
C07205=1117.752,-6.813,-50.721,179.709,6.272,149.222
C07206=1117.746,-6.564,-50.734,179.709,6.277,149.222
C07207=1117.742,-6.314,-50.748,179.710,6.281,149.223
C07208=1117.736,-6.065,-50.761,179.711,6.286,149.224
C07209=1117.731,-5.815,-50.775,179.711,6.290,149.225
C07210=1117.726,-5.566,-50.788,179.712,6.295,149.226
C07211=1117.721,-5.316,-50.802,179.712,6.300,149.227
C07212=1117.716,-5.102,-50.814,179.713,6.303,149.227
C07213=1117.712,-4.886,-50.825,179.713,6.307,149.228
C07214=1117.707,-4.672,-50.837,179.714,6.311,149.229
C07215=1117.703,-4.456,-50.848,179.714,6.315,149.229
C07216=1117.699,-4.243,-50.860,179.715,6.318,149.230
C07217=1117.695,-4.027,-50.872,179.715,6.323,149.231
C07218=1117.690,-3.812,-50.884,179.716,6.327,149.232
C07219=1117.686,-3.597,-50.895,179.716,6.330,149.232
C07220=1117.681,-3.348,-50.909,179.717,6.335,149.233
C07221=1117.676,-3.098,-50.922,179.718,6.339,149.234
C07222=1117.671,-2.849,-50.936,179.718,6.344,149.235
C07223=1117.665,-2.600,-50.950,179.719,6.349,149.236
C07224=1117.661,-2.350,-50.963,179.719,6.353,149.236
C07225=1117.655,-2.101,-50.977,179.720,6.358,149.237
C07226=1117.650,-1.850,-50.990,179.721,6.362,149.238
C07227=1117.646,-1.601,-51.004,179.721,6.366,149.239
C07228=1117.640,-1.352,-51.018,179.722,6.371,149.240
C07229=1117.635,-1.102,-51.032,179.722,6.375,149.240
C07230=1117.629,-0.853,-51.045,179.723,6.380,149.241
C07231=1117.625,-0.603,-51.059,179.723,6.385,149.242
C07232=1117.620,-0.353,-51.073,179.724,6.389,149.243
C07233=1117.614,-0.104,-51.087,179.725,6.394,149.244
C07234=1117.609,0.146,-51.101,179.725,6.399,149.245
C07235=1117.605,0.396,-51.114,179.725,6.403,149.245
C07236=1117.599,0.645,-51.128,179.726,6.407,149.246
C07237=1117.594,0.895,-51.142,179.727,6.412,149.247
C07238=1117.589,1.144,-51.156,179.727,6.416,149.248
C07239=1117.584,1.394,-51.169,179.728,6.421,149.249
C07240=1117.579,1.643,-51.183,179.729,6.425,149.249
C07241=1117.574,1.892,-51.197,179.729,6.430,149.250
C07242=1117.569,2.142,-51.211,179.730,6.435,149.251
C07243=1117.563,2.392,-51.225,179.730,6.439,149.252
C07244=1117.559,2.642,-51.239,179.731,6.443,149.253
C07245=1117.554,2.891,-51.253,179.731,6.448,149.254
C07246=1117.549,3.141,-51.267,179.732,6.453,149.255
C07247=1117.543,3.391,-51.280,179.732,6.457,149.255
C07248=1117.538,3.640,-51.294,179.733,6.462,149.256
C07249=1117.533,3.890,-51.309,179.734,6.466,149.257
C07250=1117.528,4.139,-51.323,179.735,6.471,149.258
C07251=1117.523,4.388,-51.336,179.734,6.475,149.259
C07252=1117.518,4.638,-51.350,179.735,6.480,149.260
C07253=1117.513,4.887,-51.365,179.736,6.484,149.260
C07254=1117.507,5.137,-51.378,179.737,6.489,149.261
C07255=1117.502,5.387,-51.392,179.737,6.493,149.262
C07256=1117.497,5.636,-51.407,179.738,6.498,149.263
C07257=1117.492,5.886,-51.421,179.738,6.503,149.264
C07258=1117.487,6.135,-51.435,179.738,6.507,149.265
C07259=1117.482,6.385,-51.449,179.739,6.511,149.265
C07260=1117.477,6.635,-51.463,179.740,6.516,149.266
C07261=1117.473,6.884,-51.477,179.740,6.521,149.267
C07262=1117.467,7.133,-51.491,179.741,6.525,149.268
C07263=1117.462,7.383,-51.505,179.741,6.530,149.269
C07264=1117.457,7.632,-51.519,179.742,6.535,149.270
C07265=1117.452,7.882,-51.534,179.742,6.539,149.271
C07266=1117.447,8.131,-51.548,179.743,6.543,149.271
C07267=1117.442,8.381,-51.562,179.743,6.548,149.272
C07268=1117.438,8.596,-51.574,179.744,6.552,149.273
C07269=1117.433,8.811,-51.587,179.744,6.556,149.274
C07270=1117.429,9.025,-51.599,179.745,6.560,149.274
C07271=1117.424,9.240,-51.610,179.746,6.564,149.275
C07272=1117.420,9.455,-51.623,179.746,6.568,149.276
C07273=1117.415,9.669,-51.635,179.747,6.572,149.277
C07274=1117.411,9.884,-51.647,179.747,6.576,149.277
C07275=1117.407,10.099,-51.660,179.748,6.580,149.278
C07276=1117.401,10.348,-51.674,179.749,6.585,149.279
C07277=1117.396,10.598,-51.688,179.749,6.589,149.280
C07278=1117.391,10.848,-51.702,179.750,6.594,149.281
C07279=1117.386,11.097,-51.717,179.751,6.598,149.281
C07280=1117.382,11.347,-51.732,179.751,6.603,149.282
C07281=1117.377,11.596,-51.746,179.752,6.608,149.283
C07282=1117.371,11.845,-51.760,179.753,6.612,149.284
C07283=1117.366,12.095,-51.774,179.753,6.617,149.285
C07284=1117.361,12.345,-51.788,179.754,6.621,149.285
C07285=1117.356,12.594,-51.803,179.755,6.626,149.286
C07286=1117.351,12.844,-51.818,179.756,6.630,149.287
C07287=1117.347,13.093,-51.832,179.756,6.635,149.288
C07288=1117.342,13.343,-51.846,179.757,6.640,149.288
C07289=1117.335,13.592,-51.861,179.758,6.644,149.289
C07290=1117.330,13.842,-51.875,179.758,6.648,149.290
C07291=1117.325,14.092,-51.889,179.759,6.652,149.291
C07292=1117.321,14.341,-51.904,179.759,6.657,149.292
C07293=1117.316,14.590,-51.919,179.760,6.662,149.292
C07294=1117.311,14.840,-51.933,179.761,6.666,149.293
C07295=1117.306,15.090,-51.947,179.762,6.671,149.294
C07296=1117.300,15.339,-51.963,179.762,6.675,149.295
C07297=1117.296,15.589,-51.977,179.763,6.680,149.296
C07298=1117.290,15.838,-51.991,179.764,6.684,149.296
C07299=1117.285,16.087,-52.006,179.765,6.689,149.297
C07300=1117.280,16.337,-52.020,179.766,6.693,149.298
C07301=1117.275,16.587,-52.034,179.766,6.698,149.299
C07302=1117.270,16.836,-52.050,179.767,6.702,149.299
